//展开工位
expand_initialization_OK:=FALSE;
Expand_Group_clean_OK:=FALSE;
Expand_up_liquid_OK:=FALSE;
Expand_silica_gel_plate_OK:=FALSE;
展缸1气缸1手动:=FALSE;
展缸1气缸1自动:=FALSE;
展缸1进液电池阀1手动:=FALSE;
展缸1进液电池阀1自动:=FALSE;
展缸1排液电池阀1手动:=FALSE;
展缸1排液电池阀1自动:=FALSE;
展缸1吹气电池阀1手动:=FALSE;
展缸1吹气电池阀1自动:=FALSE;
展缸1气缸2手动:=FALSE;
展缸1气缸2自动:=FALSE;
展缸1进液电池阀2手动:=FALSE;
展缸1进液电池阀2自动:=FALSE;
展缸1排液电池阀2手动:=FALSE;
展缸1排液电池阀2自动:=FALSE;
展缸1吹气电池阀2手动:=FALSE;
展缸1吹气电池阀2自动:=FALSE;
展缸1气缸3手动:=FALSE;
展缸1气缸3自动:=FALSE;
展缸1进液电池阀3手动:=FALSE;
展缸1进液电池阀3自动:=FALSE;	
展缸1排液电池阀3手动:=FALSE;
展缸1排液电池阀3自动:=FALSE;
展缸1吹气电池阀3手动:=FALSE;
展缸1吹气电池阀3自动:=FALSE;
展缸1气缸4手动:=FALSE;
展缸1气缸4自动:=FALSE;
展缸1进液电池阀4手动:=FALSE;
展缸1进液电池阀4自动:=FALSE;	
展缸1排液电池阀4手动:=FALSE;
展缸1排液电池阀4自动:=FALSE;
展缸1吹气电池阀4手动:=FALSE;
展缸1吹气电池阀4自动:=FALSE;
展缸2气缸1手动:=FALSE;
展缸2气缸1自动:=FALSE;
展缸2进液电池阀1手动:=FALSE;
展缸2进液电池阀1自动:=FALSE;
展缸2排液电池阀1手动:=FALSE;
展缸2排液电池阀1自动:=FALSE;
展缸2吹气电池阀1手动:=FALSE;
展缸2吹气电池阀1自动:=FALSE;
展缸2气缸2手动:=FALSE;
展缸2气缸2自动:=FALSE;
展缸2进液电池阀2手动:=FALSE;
展缸2进液电池阀2自动:=FALSE;
展缸2排液电池阀2手动:=FALSE;
展缸2排液电池阀2自动:=FALSE;
展缸2吹气电池阀2手动:=FALSE;
展缸2吹气电池阀2自动:=FALSE;
展缸2气缸3手动:=FALSE;
展缸2气缸3自动:=FALSE;
展缸2进液电池阀3手动:=FALSE;
展缸2进液电池阀3自动:=FALSE;	
展缸2排液电池阀3手动:=FALSE;
展缸2排液电池阀3自动:=FALSE;
展缸2吹气电池阀3手动:=FALSE;
展缸2吹气电池阀3自动:=FALSE;
展缸2气缸4手动:=FALSE;
展缸2气缸4自动:=FALSE;
展缸2进液电池阀4手动:=FALSE;
展缸2进液电池阀4自动:=FALSE;	
展缸2排液电池阀4手动:=FALSE;
展缸2排液电池阀4自动:=FALSE;
展缸2吹气电池阀4手动:=FALSE;
展缸2吹气电池阀4自动:=FALSE;
Expand_Step:=0;
//拍照刮板
刮板拍照真空自动:=FALSE;
刮板拍照真空手动:=FALSE;
刮板拍照无刷电机手动:=FALSE;
刮板拍照无刷电机自动:=FALSE;
刮板拍照定位气缸手动:=FALSE;
刮板拍照定位气缸自动:=FALSE;
粉末收集器定位手动:=FALSE;
粉末收集器定位自动:=FALSE;
刮板拍照遮光气缸手动:=FALSE;
刮板拍照遮光气缸自动:=FALSE;
刮板拍照旋转气缸手动:=FALSE;
刮板拍照旋转气缸自动:=FALSE;
刮板拍照下压气缸手动:=FALSE;
刮板拍照下压气缸自动:=FALSE;
 scrape_IsLast := FALSE;       // ★ 新增		
scrape_PhotoMode:=0;
scrape_Step:=0;
Camera_scraper_initialization_OK:=FALSE;
Photo_preparation_completed_OK:=FALSE;
Scraper_collection_completed:=FALSE;
Robot_completes_material_retrieval:=FALSE;	

//上样点样
上样定位手动:=FALSE;
上样定位自动:=FALSE;
上样点样三通电池阀手动:=FALSE;
上样点样三通电池阀自动:=FALSE;
上样吹气手动:=FALSE;
上样吹气自动:=FALSE;
打样瓶上料轴3YDATE.fAbsTarget:=0;
点样轴6XDATE.fAbsTarget:=0;
点样轴7YDATE.fAbsTarget:=0;
上样轴4X轴DATE.fAbsTarget:=0;
上样轴5Z轴DATE.fAbsTarget:=0;
点样轴7YDATE.xMoveAbs:=FALSE;
点样轴6XDATE.xMoveAbs:=FALSE;
上样轴5Z轴DATE.xMoveAbs:=FALSE;
上样轴4X轴DATE.xMoveAbs:=FALSE;
打样瓶上料轴3YDATE.xMoveAbs:=FALSE;
Sampling_Spray_sample_OK:=FALSE;
Sampling_liquid_absorption:=FALSE;
Sampling_preparation_OK:=FALSE;
大真空泵站位[11]:=FALSE;
大真空泵自动:=FALSE;
Sampling_Step:=0;

//机器人

泵站位符:=FALSE;
上样料架报警:=FALSE;
溶液收集瓶定位自动:=FALSE;
溶液收集瓶定位手动:=FALSE;
END_ACTION

END_PROGRAM

// Device/Application/40_Man/PLC_Cyinder_气缸动作
PROGRAM PLC_Cyinder_气缸动作
VAR
	cylinder_0: FB_cylinder;
	cylinder_1: FB_cylinder;
	cylinder_2: FB_cylinder;
	cylinder_3 :FB_cylinder ;
	cylinder_4 :FB_cylinder ;
	cylinder_5 :FB_cylinder ;
	cylinder_6 :FB_cylinder ;
	cylinder_7 :FB_cylinder ;
	cylinder_8 :FB_cylinder ;
	cylinder_9 :FB_cylinder ;
	cylinder_10 :FB_cylinder ;
	cylinder_11 :FB_cylinder ;
	cylinder_12 :FB_cylinder ;
	cylinder_13 :FB_cylinder ;
	cylinder_14 :FB_cylinder ;
	cylinder_15 :FB_cylinder ;
	cylinder_16 :FB_cylinder ;
	cylinder_17 :FB_cylinder ;
	cylinder_18 :FB_cylinder ;
	cylinder_19 :FB_cylinder ;
	cylinder_20 :FB_cylinder ;
	cylinder_21 :FB_cylinder ;
	cylinder_22 :FB_cylinder ;
	cylinder_23 :FB_cylinder ;
	cylinder_24 :FB_cylinder ;
	cylinder_25 :FB_cylinder ;
	cylinder_26 :FB_cylinder ;
	cylinder_27 :FB_cylinder ;
	cylinder_28 :FB_cylinder ;
	cylinder_29 :FB_cylinder ;
	cylinder_30 :FB_cylinder ;
	cylinder_31 :FB_cylinder ;
	cylinder_32 :FB_cylinder ;
	cylinder_33 :FB_cylinder ;
	cylinder_34 :FB_cylinder ;
	cylinder_35 :FB_cylinder ;
	cylinder_36 :FB_cylinder ;
	cylinder_37 :FB_cylinder ;
	cylinder_38 :FB_cylinder ;
	cylinder_39 :FB_cylinder ;
	cylinder_40 :FB_cylinder ;
	cylinder_41 :FB_cylinder ;
	cylinder_42 :FB_cylinder ;
	cylinder_43 :FB_cylinder ;
	cylinder_44 :FB_cylinder ;
	cylinder_45 :FB_cylinder ;
	cylinder_46 :FB_cylinder ;
	cylinder_47 :FB_cylinder ;
	cylinder_48 :FB_cylinder ;
	cylinder_49 :FB_cylinder ;
	cylinder_50 :FB_cylinder ;
	bDeployCommandsArmed: BOOL;
	bAnyDeployCommandRequested: BOOL;

END_VAR

// PLC deploy auxiliary-actuator gate BEGIN
bAnyDeployCommandRequested := 展缸1气缸1手动
	OR 展缸1气缸1自动
	OR 展缸1气缸2手动
	OR 展缸1气缸2自动
	OR 展缸1气缸3手动
	OR 展缸1气缸3自动
	OR 展缸1气缸4手动
	OR 展缸1气缸4自动
	OR 展缸2气缸1手动
	OR 展缸2气缸1自动
	OR 展缸2气缸2手动
	OR 展缸2气缸2自动
	OR 展缸2气缸3手动
	OR 展缸2气缸3自动
	OR 展缸2气缸4手动
	OR 展缸2气缸4自动
	OR 大真空泵手动
	OR 大真空泵自动
	OR 收集下压气缸手动
	OR 收集下压气缸自动
	OR 收集夹持气缸手动
	OR 收集夹持气缸自动
	OR 收集升降气缸手动
	OR 收集升降气缸自动
	OR 收集伸缩气缸手动
	OR 收集伸缩气缸自动
	OR 刮板拍照遮光气缸手动
	OR 刮板拍照遮光气缸自动
	OR 刮板拍照旋转气缸手动
	OR 刮板拍照旋转气缸自动
	OR 刮板拍照下压气缸手动
	OR 刮板拍照下压气缸自动
	OR 展缸1进液电池阀1手动
	OR 展缸1进液电池阀1自动
	OR 展缸1进液电池阀2手动
	OR 展缸1进液电池阀2自动
	OR 展缸1进液电池阀3手动
	OR 展缸1进液电池阀3自动
	OR 展缸1进液电池阀4手动
	OR 展缸1进液电池阀4自动
	OR 展缸1排液电池阀1手动
	OR 展缸1排液电池阀1自动
	OR 展缸1排液电池阀2手动
	OR 展缸1排液电池阀2自动
	OR 展缸1排液电池阀3手动
	OR 展缸1排液电池阀3自动
	OR 展缸1排液电池阀4手动
	OR 展缸1排液电池阀4自动
	OR 展缸1吹气电池阀1手动
	OR 展缸1吹气电池阀1自动
	OR 展缸1吹气电池阀2手动
	OR 展缸1吹气电池阀2自动
	OR 展缸1吹气电池阀3手动
	OR 展缸1吹气电池阀3自动
	OR 展缸1吹气电池阀4手动
	OR 展缸1吹气电池阀4自动
	OR 展缸2进液电池阀1手动
	OR 展缸2进液电池阀1自动
	OR 展缸2进液电池阀2手动
	OR 展缸2进液电池阀2自动
	OR 展缸2进液电池阀3手动
	OR 展缸2进液电池阀3自动
	OR 展缸2进液电池阀4手动
	OR 展缸2进液电池阀4自动
	OR 展缸2排液电池阀1手动
	OR 展缸2排液电池阀1自动
	OR 展缸2排液电池阀2手动
	OR 展缸2排液电池阀2自动
	OR 展缸2排液电池阀3手动
	OR 展缸2排液电池阀3自动
	OR 展缸2排液电池阀4手动
	OR 展缸2排液电池阀4自动
	OR 展缸2吹气电池阀1手动
	OR 展缸2吹气电池阀1自动
	OR 展缸2吹气电池阀2手动
	OR 展缸2吹气电池阀2自动
	OR 展缸2吹气电池阀3手动
	OR 展缸2吹气电池阀3自动
	OR 展缸2吹气电池阀4手动
	OR 展缸2吹气电池阀4自动
	OR 收集进液手动
	OR 收集进液自动
	OR 收集排液手动
	OR 收集排液自动
	OR 收集正压排液手动
	OR 收集正压排液自动
	OR 溶液收集瓶定位手动
	OR 溶液收集瓶定位自动
	OR 上样定位手动
	OR 上样定位自动
	OR 上样点样三通电池阀手动
	OR 上样点样三通电池阀自动
	OR 刮板拍照真空手动
	OR 刮板拍照真空自动
	OR 刮板拍照无刷电机手动
	OR 刮板拍照无刷电机自动
	OR 刮板拍照定位气缸手动
	OR 刮板拍照定位气缸自动
	OR 粉末收集器定位手动
	OR 粉末收集器定位自动
	OR 上样吹气手动
	OR 上样吹气自动;
IF ((NOT PLC_Ready) OR ((PLC_Deploy_State<>0) AND (PLC_Deploy_State<>30))) THEN
	bDeployCommandsArmed := FALSE;
ELSIF NOT bAnyDeployCommandRequested THEN
	// A command written while maintenance was active must first return FALSE;
	// it is never replayed automatically when the maintenance lock is released.
	bDeployCommandsArmed := TRUE;
END_IF
// PLC deploy auxiliary-actuator gate END
//气缸动作
//展缸1气缸1
cylinder_0(
    xManualRetract := , 
    xAutoRetract := , 
    yValve2 => , 
    cylinder_type := 0, 

	xManualAuto:=ManualAuto  , 
	xManualExtend:=PLC_Ready AND ((PLC_Deploy_State=0) OR (PLC_Deploy_State=30)) AND bDeployCommandsArmed AND (展缸1气缸1手动), 
	xAutoExtend:= PLC_Ready AND ((PLC_Deploy_State=0) OR (PLC_Deploy_State=30)) AND bDeployCommandsArmed AND (展缸1气缸1自动), 
	xReset:=复位  , 
	xPosExtend:= 展缸1气缸1原点, 
	xPosRetract:= 展缸1气缸1动点 , 
	tTimeout:= T#5S, 
	yValve1=> 展缸1气缸1 , 
	bAlarm=> cyinderAlarm.0);
//展缸1气缸2
cylinder_1(
    xManualRetract := , 
    xAutoRetract := , 
    yValve2 => , 
    cylinder_type :=0 , 

	xManualAuto:=ManualAuto  , 
	xManualExtend:=PLC_Ready AND ((PLC_Deploy_State=0) OR (PLC_Deploy_State=30)) AND bDeployCommandsArmed AND (展缸1气缸2手动), 
	xAutoExtend:= PLC_Ready AND ((PLC_Deploy_State=0) OR (PLC_Deploy_State=30)) AND bDeployCommandsArmed AND (展缸1气缸2自动), 
	xReset:=复位  , 
	xPosExtend:= 展缸1气缸2原点, 
	xPosRetract:= 展缸1气缸2动点 , 
	tTimeout:= T#5S, 
	yValve1=> 展缸1气缸2, 
	bAlarm=> cyinderAlarm.1);
//展缸1气缸3
cylinder_2(
    xManualRetract := , 
    xAutoRetract := , 
    yValve2 => , 
    cylinder_type := 0, 

	xManualAuto:=ManualAuto  , 
	xManualExtend:=PLC_Ready AND ((PLC_Deploy_State=0) OR (PLC_Deploy_State=30)) AND bDeployCommandsArmed AND (展缸1气缸3手动), 
	xAutoExtend:= PLC_Ready AND ((PLC_Deploy_State=0) OR (PLC_Deploy_State=30)) AND bDeployCommandsArmed AND (展缸1气缸3自动), 
	xReset:=复位  , 
	xPosExtend:= 展缸1气缸3原点, 
	xPosRetract:= 展缸1气缸3动点 , 
	tTimeout:= T#5S, 
	yValve1=> 展缸1气缸3, 
	bAlarm=> cyinderAlarm.2);
//展缸1气缸4
cylinder_3(
    xManualRetract := , 
    xAutoRetract := , 
    yValve2 => , 
    cylinder_type :=0 , 

	xManualAuto:=ManualAuto  , 
	xManualExtend:=PLC_Ready AND ((PLC_Deploy_State=0) OR (PLC_Deploy_State=30)) AND bDeployCommandsArmed AND (展缸1气缸4手动), 
	xAutoExtend:= PLC_Ready AND ((PLC_Deploy_State=0) OR (PLC_Deploy_State=30)) AND bDeployCommandsArmed AND (展缸1气缸4自动), 
	xReset:=复位  , 
	xPosExtend:= 展缸1气缸4原点, 
	xPosRetract:= 展缸1气缸4动点 , 
	tTimeout:= T#5S, 
	yValve1=> 展缸1气缸4, 
	bAlarm=> cyinderAlarm.3);
//展缸2气缸1
cylinder_4(
    xManualRetract := , 
    xAutoRetract := , 
    yValve2 => , 
    cylinder_type := 0, 

	xManualAuto:=ManualAuto  , 
	xManualExtend:=PLC_Ready AND ((PLC_Deploy_State=0) OR (PLC_Deploy_State=30)) AND bDeployCommandsArmed AND (展缸2气缸1手动), 
	xAutoExtend:= PLC_Ready AND ((PLC_Deploy_State=0) OR (PLC_Deploy_State=30)) AND bDeployCommandsArmed AND (展缸2气缸1自动), 
	xReset:=复位  , 
	xPosExtend:= 展缸2气缸1原点, 
	xPosRetract:= 展缸2气缸1动点 , 
	tTimeout:= T#5S, 
	yValve1=> 展缸2气缸1, 
	bAlarm=> cyinderAlarm.4);
//展缸2气缸2
cylinder_5(
    xManualRetract := , 
    xAutoRetract := , 
    yValve2 => , 
    cylinder_type :=0 , 

	xManualAuto:=ManualAuto  , 
	xManualExtend:=PLC_Ready AND ((PLC_Deploy_State=0) OR (PLC_Deploy_State=30)) AND bDeployCommandsArmed AND (展缸2气缸2手动), 
	xAutoExtend:= PLC_Ready AND ((PLC_Deploy_State=0) OR (PLC_Deploy_State=30)) AND bDeployCommandsArmed AND (展缸2气缸2自动), 
	xReset:=复位  , 
	xPosExtend:= 展缸2气缸2原点, 
	xPosRetract:= 展缸2气缸2动点 , 
	tTimeout:= T#5S, 
	yValve1=> 展缸2气缸2, 
	bAlarm=> cyinderAlarm.5);
//展缸2气缸3
cylinder_6(
    xManualRetract := , 
    xAutoRetract := , 
    yValve2 => , 
    cylinder_type := 0, 

	xManualAuto:=ManualAuto  , 
	xManualExtend:=PLC_Ready AND ((PLC_Deploy_State=0) OR (PLC_Deploy_State=30)) AND bDeployCommandsArmed AND (展缸2气缸3手动), 
	xAutoExtend:= PLC_Ready AND ((PLC_Deploy_State=0) OR (PLC_Deploy_State=30)) AND bDeployCommandsArmed AND (展缸2气缸3自动), 
	xReset:=复位  , 
	xPosExtend:= 展缸2气缸3原点, 
	xPosRetract:= 展缸2气缸3动点 , 
	tTimeout:= T#5S, 
	yValve1=> 展缸2气缸3, 
	bAlarm=> cyinderAlarm.6);
//展缸2气缸4
cylinder_7(
    xManualRetract := , 
    xAutoRetract := , 
    yValve2 => , 
    cylinder_type := 0, 

	xManualAuto:=ManualAuto  , 
	xManualExtend:=PLC_Ready AND ((PLC_Deploy_State=0) OR (PLC_Deploy_State=30)) AND bDeployCommandsArmed AND (展缸2气缸4手动), 
	xAutoExtend:= PLC_Ready AND ((PLC_Deploy_State=0) OR (PLC_Deploy_State=30)) AND bDeployCommandsArmed AND (展缸2气缸4自动), 
	xReset:=复位  , 
	xPosExtend:= 展缸2气缸4原点, 
	xPosRetract:= 展缸2气缸4动点 , 
	tTimeout:= T#5S, 
	yValve1=> 展缸2气缸4, 
	bAlarm=> cyinderAlarm.7);
//大真空泵
cylinder_8(
    xManualRetract := , 
    xAutoRetract := , 
    yValve2 => , 
    cylinder_type :=0 , 

	xManualAuto:=ManualAuto  , 
	xManualExtend:= PLC_Ready AND ((PLC_Deploy_State=0) OR (PLC_Deploy_State=30)) AND bDeployCommandsArmed AND (大真空泵手动), 
	xAutoExtend:= PLC_Ready AND ((PLC_Deploy_State=0) OR (PLC_Deploy_State=30)) AND bDeployCommandsArmed AND (大真空泵自动), 
	xReset:=复位  , 
	xPosExtend:= , 
	xPosRetract:=  , 
	tTimeout:= , 
	yValve1=> 大真空泵, 
	bAlarm=> );
//收集平台下压气缸
cylinder_9(
    xManualRetract := , 
    xAutoRetract := , 
    yValve2 => , 
    cylinder_type := 0, 

	xManualAuto:=ManualAuto  , 
	xManualExtend:= PLC_Ready AND ((PLC_Deploy_State=0) OR (PLC_Deploy_State=30)) AND bDeployCommandsArmed AND (收集下压气缸手动), 
	xAutoExtend:= PLC_Ready AND ((PLC_Deploy_State=0) OR (PLC_Deploy_State=30)) AND bDeployCommandsArmed AND (收集下压气缸自动), 
	xReset:=复位  , 
	xPosExtend:=收集平台下压气缸原点 , 
	xPosRetract:= 收集下压气缸手动 OR 收集下压气缸自动, 
	tTimeout:= T#5S, 
	yValve1=> 收集下压气缸 , 
	bAlarm=> cyinderAlarm.8);
//收集平台夹持气缸
cylinder_10(
    xManualRetract := , 
    xAutoRetract := , 
    yValve2 => , 
    cylinder_type := 0, 

	xManualAuto:=ManualAuto  , 
	xManualExtend:= PLC_Ready AND ((PLC_Deploy_State=0) OR (PLC_Deploy_State=30)) AND bDeployCommandsArmed AND (收集夹持气缸手动), 
	xAutoExtend:= PLC_Ready AND ((PLC_Deploy_State=0) OR (PLC_Deploy_State=30)) AND bDeployCommandsArmed AND (收集夹持气缸自动), 
	xReset:=复位  , 
	xPosExtend:=收集平台夹持气缸原点 , 
	xPosRetract:= 收集平台夹持气缸动点, 
	tTimeout:= T#5S, 
	yValve1=> 收集夹持气缸  , 
	bAlarm=> cyinderAlarm.9);	
//收集平台升降气缸
cylinder_11(
    xManualRetract := , 
    xAutoRetract := , 
    yValve2 => , 
    cylinder_type := 0, 

	xManualAuto:=ManualAuto  , 
	xManualExtend:= PLC_Ready AND ((PLC_Deploy_State=0) OR (PLC_Deploy_State=30)) AND bDeployCommandsArmed AND (收集升降气缸手动), 
	xAutoExtend:= PLC_Ready AND ((PLC_Deploy_State=0) OR (PLC_Deploy_State=30)) AND bDeployCommandsArmed AND (收集升降气缸自动), 
	xReset:=复位  , 
	xPosExtend:=收集平台升降气缸原点 , 
	xPosRetract:= 收集平台升降气缸动点, 
	tTimeout:= T#5S, 
	yValve1=> 收集升降气缸   , 
	bAlarm=> cyinderAlarm.10);	
//收集平台伸缩气缸
cylinder_12(
    xManualRetract := , 
    xAutoRetract := , 
    yValve2 => , 
    cylinder_type :=0 , 

	xManualAuto:=ManualAuto  , 
	xManualExtend:= PLC_Ready AND ((PLC_Deploy_State=0) OR (PLC_Deploy_State=30)) AND bDeployCommandsArmed AND (收集伸缩气缸手动), 
	xAutoExtend:= PLC_Ready AND ((PLC_Deploy_State=0) OR (PLC_Deploy_State=30)) AND bDeployCommandsArmed AND (收集伸缩气缸自动), 
	xReset:=复位, 
	xPosExtend:=收集平台推出气缸原点, 
	xPosRetract:= 收集平台推出气缸动点, 
	tTimeout:= T#5S, 
	yValve1=> 收集伸缩气缸, 
	bAlarm=> cyinderAlarm.11);		
//刮板拍照遮光气缸
cylinder_13(
    xManualRetract := , 
    xAutoRetract := , 
    yValve2 => , 
    cylinder_type :=0 , 

	xManualAuto:=ManualAuto  , 
	xManualExtend:= PLC_Ready AND ((PLC_Deploy_State=0) OR (PLC_Deploy_State=30)) AND bDeployCommandsArmed AND (刮板拍照遮光气缸手动), 
	xAutoExtend:=PLC_Ready AND ((PLC_Deploy_State=0) OR (PLC_Deploy_State=30)) AND bDeployCommandsArmed AND (刮板拍照遮光气缸自动), 
	xReset:=复位  , 
	xPosExtend:=刮板拍照遮光气缸上位 , 
	xPosRetract:= 刮板拍照遮光气缸下位, 
	tTimeout:= T#5S, 
	yValve1=>  刮板拍照遮光气缸, 
	bAlarm=> cyinderAlarm.12);		
//刮板拍照旋转气缸
cylinder_14(
    xManualRetract := , 
    xAutoRetract := , 
    yValve2 => , 
    cylinder_type := 0, 

	xManualAuto:=ManualAuto  , 
	xManualExtend:= PLC_Ready AND ((PLC_Deploy_State=0) OR (PLC_Deploy_State=30)) AND bDeployCommandsArmed AND (刮板拍照旋转气缸手动 AND 刮板轴9XDATE.fActPos>330), 
	xAutoExtend:=PLC_Ready AND ((PLC_Deploy_State=0) OR (PLC_Deploy_State=30)) AND bDeployCommandsArmed AND (刮板拍照旋转气缸自动), 
	xReset:=复位  , 
	xPosExtend:=刮板拍照旋转气缸原点  , 
	xPosRetract:= 刮板拍照旋转气缸动点, 
	tTimeout:= T#5S, 
	yValve1=>  刮板拍照旋转气缸   , 
	bAlarm=> cyinderAlarm.13);		
//刮板拍照下压气缸
cylinder_15(
    xManualRetract := , 
    xAutoRetract := , 
    yValve2 => , 
    cylinder_type := 0, 

	xManualAuto:=ManualAuto  , 
	xManualExtend:= PLC_Ready AND ((PLC_Deploy_State=0) OR (PLC_Deploy_State=30)) AND bDeployCommandsArmed AND (刮板拍照下压气缸手动), 
	xAutoExtend:=PLC_Ready AND ((PLC_Deploy_State=0) OR (PLC_Deploy_State=30)) AND bDeployCommandsArmed AND (刮板拍照下压气缸自动), 
	xReset:=复位  , 
	xPosExtend:=刮板拍照下压气缸上位, 
	xPosRetract:=刮板拍照下压气缸手动 OR 刮板拍照下压气缸自动 , 
	tTimeout:= T#5S, 
	yValve1=>  刮板拍照下压气缸, 
	bAlarm=> cyinderAlarm.14);
//展缸1进液电池阀1
cylinder_17(
    xManualRetract := , 
    xAutoRetract := , 
    yValve2 => , 
    cylinder_type :=0 , 

	xManualAuto:=ManualAuto  , 
	xManualExtend:= PLC_Ready AND ((PLC_Deploy_State=0) OR (PLC_Deploy_State=30)) AND bDeployCommandsArmed AND (展缸1进液电池阀1手动), 
	xAutoExtend:= PLC_Ready AND ((PLC_Deploy_State=0) OR (PLC_Deploy_State=30)) AND bDeployCommandsArmed AND (展缸1进液电池阀1自动), 
	xReset:=复位  , 
	xPosExtend:=   , 
	xPosRetract:= , 
	tTimeout:= , 
	yValve1=> 展缸1进液电池阀1, 
	bAlarm=> );	
//展缸1进液电池阀2
cylinder_18(
    xManualRetract := , 
    xAutoRetract := , 
    yValve2 => , 
    cylinder_type := 0, 

	xManualAuto:=ManualAuto  , 
	xManualExtend:= PLC_Ready AND ((PLC_Deploy_State=0) OR (PLC_Deploy_State=30)) AND bDeployCommandsArmed AND (展缸1进液电池阀2手动), 
	xAutoExtend:= PLC_Ready AND ((PLC_Deploy_State=0) OR (PLC_Deploy_State=30)) AND bDeployCommandsArmed AND (展缸1进液电池阀2自动), 
	xReset:=复位  , 
	xPosExtend:=   , 
	xPosRetract:= , 
	tTimeout:= , 
	yValve1=> 展缸1进液电池阀2, 
	bAlarm=> );	
//展缸1进液电池阀3
cylinder_19(
    xManualRetract := , 
    xAutoRetract := , 
    yValve2 => , 
    cylinder_type := 0, 

	xManualAuto:=ManualAuto  , 
	xManualExtend:= PLC_Ready AND ((PLC_Deploy_State=0) OR (PLC_Deploy_State=30)) AND bDeployCommandsArmed AND (展缸1进液电池阀3手动), 
	xAutoExtend:= PLC_Ready AND ((PLC_Deploy_State=0) OR (PLC_Deploy_State=30)) AND bDeployCommandsArmed AND (展缸1进液电池阀3自动), 
	xReset:=复位  , 
	xPosExtend:=   , 
	xPosRetract:= , 
	tTimeout:= , 
	yValve1=> 展缸1进液电池阀3, 
	bAlarm=> );	
//展缸1进液电池阀4
cylinder_20(
    xManualRetract := , 
    xAutoRetract := , 
    yValve2 => , 
    cylinder_type := 0, 

	xManualAuto:=ManualAuto  , 
	xManualExtend:= PLC_Ready AND ((PLC_Deploy_State=0) OR (PLC_Deploy_State=30)) AND bDeployCommandsArmed AND (展缸1进液电池阀4手动), 
	xAutoExtend:= PLC_Ready AND ((PLC_Deploy_State=0) OR (PLC_Deploy_State=30)) AND bDeployCommandsArmed AND (展缸1进液电池阀4自动), 
	xReset:=复位  , 
	xPosExtend:=   , 
	xPosRetract:= , 
	tTimeout:= , 
	yValve1=> 展缸1进液电池阀4, 
	bAlarm=> );	
//展缸1排液电池阀1
cylinder_21(
    xManualRetract := , 
    xAutoRetract := , 
    yValve2 => , 
    cylinder_type := 0, 

	xManualAuto:=ManualAuto  , 
	xManualExtend:= PLC_Ready AND ((PLC_Deploy_State=0) OR (PLC_Deploy_State=30)) AND bDeployCommandsArmed AND (展缸1排液电池阀1手动), 
	xAutoExtend:= PLC_Ready AND ((PLC_Deploy_State=0) OR (PLC_Deploy_State=30)) AND bDeployCommandsArmed AND (展缸1排液电池阀1自动), 
	xReset:=复位  , 
	xPosExtend:=   , 
	xPosRetract:= , 
	tTimeout:= , 
	yValve1=> 展缸1排液电池阀1, 
	bAlarm=> );	
//展缸1排液电池阀2
cylinder_22(
    xManualRetract := , 
    xAutoRetract := , 
    yValve2 => , 
    cylinder_type :=0 , 

	xManualAuto:=ManualAuto  , 
	xManualExtend:= PLC_Ready AND ((PLC_Deploy_State=0) OR (PLC_Deploy_State=30)) AND bDeployCommandsArmed AND (展缸1排液电池阀2手动), 
	xAutoExtend:= PLC_Ready AND ((PLC_Deploy_State=0) OR (PLC_Deploy_State=30)) AND bDeployCommandsArmed AND (展缸1排液电池阀2自动), 
	xReset:=复位  , 
	xPosExtend:=   , 
	xPosRetract:= , 
	tTimeout:= , 
	yValve1=> 展缸1排液电池阀2, 
	bAlarm=> );	
//展缸1排液电池阀3
cylinder_23(
    xManualRetract := , 
    xAutoRetract := , 
    yValve2 => , 
    cylinder_type :=0 , 

	xManualAuto:=ManualAuto, 
	xManualExtend:= PLC_Ready AND ((PLC_Deploy_State=0) OR (PLC_Deploy_State=30)) AND bDeployCommandsArmed AND (展缸1排液电池阀3手动), 
	xAutoExtend:= PLC_Ready AND ((PLC_Deploy_State=0) OR (PLC_Deploy_State=30)) AND bDeployCommandsArmed AND (展缸1排液电池阀3自动), 
	xReset:=复位  , 
	xPosExtend:=   , 
	xPosRetract:= , 
	tTimeout:= , 
	yValve1=> 展缸1排液电池阀3, 
	bAlarm=> );	
//展缸1排液电池阀4
cylinder_24(
    xManualRetract := , 
    xAutoRetract := , 
    yValve2 => , 
    cylinder_type := 0, 

	xManualAuto:=ManualAuto, 
	xManualExtend:= PLC_Ready AND ((PLC_Deploy_State=0) OR (PLC_Deploy_State=30)) AND bDeployCommandsArmed AND (展缸1排液电池阀4手动), 
	xAutoExtend:= PLC_Ready AND ((PLC_Deploy_State=0) OR (PLC_Deploy_State=30)) AND bDeployCommandsArmed AND (展缸1排液电池阀4自动), 
	xReset:=复位  , 
	xPosExtend:=   , 
	xPosRetract:= , 
	tTimeout:= , 
	yValve1=> 展缸1排液电池阀4, 
	bAlarm=> );	
//展缸1吹气电池阀1
cylinder_25(
    xManualRetract := , 
    xAutoRetract := , 
    yValve2 => , 
    cylinder_type := 0, 

	xManualAuto:=ManualAuto, 
	xManualExtend:= PLC_Ready AND ((PLC_Deploy_State=0) OR (PLC_Deploy_State=30)) AND bDeployCommandsArmed AND (展缸1吹气电池阀1手动), 
	xAutoExtend:= PLC_Ready AND ((PLC_Deploy_State=0) OR (PLC_Deploy_State=30)) AND bDeployCommandsArmed AND (展缸1吹气电池阀1自动), 
	xReset:=复位  , 
	xPosExtend:=   , 
	xPosRetract:= , 
	tTimeout:= , 
	yValve1=> 展缸1吹气电池阀1, 
	bAlarm=> );	
//展缸1吹气电池阀2
cylinder_26(
    xManualRetract := , 
    xAutoRetract := , 
    yValve2 => , 
    cylinder_type := 0, 

	xManualAuto:=ManualAuto, 
	xManualExtend:= PLC_Ready AND ((PLC_Deploy_State=0) OR (PLC_Deploy_State=30)) AND bDeployCommandsArmed AND (展缸1吹气电池阀2手动), 
	xAutoExtend:= PLC_Ready AND ((PLC_Deploy_State=0) OR (PLC_Deploy_State=30)) AND bDeployCommandsArmed AND (展缸1吹气电池阀2自动), 
	xReset:=复位  , 
	xPosExtend:=   , 
	xPosRetract:= , 
	tTimeout:= , 
	yValve1=> 展缸1吹气电池阀2, 
	bAlarm=> );	
//展缸1吹气电池阀3
cylinder_27(
    xManualRetract := , 
    xAutoRetract := , 
    yValve2 => , 
    cylinder_type := 0, 

	xManualAuto:=ManualAuto  , 
	xManualExtend:= PLC_Ready AND ((PLC_Deploy_State=0) OR (PLC_Deploy_State=30)) AND bDeployCommandsArmed AND (展缸1吹气电池阀3手动), 
	xAutoExtend:= PLC_Ready AND ((PLC_Deploy_State=0) OR (PLC_Deploy_State=30)) AND bDeployCommandsArmed AND (展缸1吹气电池阀3自动), 
	xReset:=复位  , 
	xPosExtend:=   , 
	xPosRetract:= , 
	tTimeout:= , 
	yValve1=> 展缸1吹气电池阀3, 
	bAlarm=> );	
//展缸1吹气电池阀4
cylinder_28(
    xManualRetract := , 
    xAutoRetract := , 
    yValve2 => , 
    cylinder_type := 0, 

	xManualAuto:=ManualAuto, 
	xManualExtend:= PLC_Ready AND ((PLC_Deploy_State=0) OR (PLC_Deploy_State=30)) AND bDeployCommandsArmed AND (展缸1吹气电池阀4手动), 
	xAutoExtend:= PLC_Ready AND ((PLC_Deploy_State=0) OR (PLC_Deploy_State=30)) AND bDeployCommandsArmed AND (展缸1吹气电池阀4自动), 
	xReset:=复位  , 
	xPosExtend:=   , 
	xPosRetract:= , 
	tTimeout:= , 
	yValve1=> 展缸1吹气电池阀4, 
	bAlarm=> );	
//展缸2进液电池阀1
cylinder_29(
    xManualRetract := , 
    xAutoRetract := , 
    yValve2 => , 
    cylinder_type := 0, 

	xManualAuto:=ManualAuto, 
	xManualExtend:= PLC_Ready AND ((PLC_Deploy_State=0) OR (PLC_Deploy_State=30)) AND bDeployCommandsArmed AND (展缸2进液电池阀1手动), 
	xAutoExtend:= PLC_Ready AND ((PLC_Deploy_State=0) OR (PLC_Deploy_State=30)) AND bDeployCommandsArmed AND (展缸2进液电池阀1自动), 
	xReset:=复位  , 
	xPosExtend:=   , 
	xPosRetract:= , 
	tTimeout:= , 
	yValve1=> 展缸2进液电池阀1, 
	bAlarm=> );	
//展缸2进液电池阀2
cylinder_30(
    xManualRetract := , 
    xAutoRetract := , 
    yValve2 => , 
    cylinder_type := 0, 

	xManualAuto:=ManualAuto, 
	xManualExtend:= PLC_Ready AND ((PLC_Deploy_State=0) OR (PLC_Deploy_State=30)) AND bDeployCommandsArmed AND (展缸2进液电池阀2手动), 
	xAutoExtend:= PLC_Ready AND ((PLC_Deploy_State=0) OR (PLC_Deploy_State=30)) AND bDeployCommandsArmed AND (展缸2进液电池阀2自动), 
	xReset:=复位  , 
	xPosExtend:=   , 
	xPosRetract:= , 
	tTimeout:= , 
	yValve1=> 展缸2进液电池阀2, 
	bAlarm=> );	
//展缸2进液电池阀3
cylinder_31(
    xManualRetract := , 
    xAutoRetract := , 
    yValve2 => , 
    cylinder_type := 0, 

	xManualAuto:=ManualAuto, 
	xManualExtend:= PLC_Ready AND ((PLC_Deploy_State=0) OR (PLC_Deploy_State=30)) AND bDeployCommandsArmed AND (展缸2进液电池阀3手动), 
	xAutoExtend:= PLC_Ready AND ((PLC_Deploy_State=0) OR (PLC_Deploy_State=30)) AND bDeployCommandsArmed AND (展缸2进液电池阀3自动), 
	xReset:=复位  , 
	xPosExtend:=   , 
	xPosRetract:= , 
	tTimeout:= , 
	yValve1=> 展缸2进液电池阀3, 
	bAlarm=> );	
//展缸2进液电池阀4
cylinder_32(
    xManualRetract := , 
    xAutoRetract := , 
    yValve2 => , 
    cylinder_type := 0, 

	xManualAuto:=ManualAuto, 
	xManualExtend:= PLC_Ready AND ((PLC_Deploy_State=0) OR (PLC_Deploy_State=30)) AND bDeployCommandsArmed AND (展缸2进液电池阀4手动), 
	xAutoExtend:= PLC_Ready AND ((PLC_Deploy_State=0) OR (PLC_Deploy_State=30)) AND bDeployCommandsArmed AND (展缸2进液电池阀4自动), 
	xReset:=复位  , 
	xPosExtend:=   , 
	xPosRetract:= , 
	tTimeout:= , 
	yValve1=> 展缸2进液电池阀4, 
	bAlarm=> );	
//展缸2排液电池阀1
cylinder_33(
    xManualRetract := , 
    xAutoRetract := , 
    yValve2 => , 
    cylinder_type := 0, 

	xManualAuto:=ManualAuto, 
	xManualExtend:= PLC_Ready AND ((PLC_Deploy_State=0) OR (PLC_Deploy_State=30)) AND bDeployCommandsArmed AND (展缸2排液电池阀1手动), 
	xAutoExtend:= PLC_Ready AND ((PLC_Deploy_State=0) OR (PLC_Deploy_State=30)) AND bDeployCommandsArmed AND (展缸2排液电池阀1自动), 
	xReset:=复位  , 
	xPosExtend:=   , 
	xPosRetract:= , 
	tTimeout:= , 
	yValve1=> 展缸2排液电池阀1, 
	bAlarm=> );	
//展缸2排液电池阀2
cylinder_34(
    xManualRetract := , 
    xAutoRetract := , 
    yValve2 => , 
    cylinder_type := 0, 

	xManualAuto:=ManualAuto, 
	xManualExtend:= PLC_Ready AND ((PLC_Deploy_State=0) OR (PLC_Deploy_State=30)) AND bDeployCommandsArmed AND (展缸2排液电池阀2手动), 
	xAutoExtend:= PLC_Ready AND ((PLC_Deploy_State=0) OR (PLC_Deploy_State=30)) AND bDeployCommandsArmed AND (展缸2排液电池阀2自动), 
	xReset:=复位  , 
	xPosExtend:=   , 
	xPosRetract:= , 
	tTimeout:= , 
	yValve1=> 展缸2排液电池阀2, 
	bAlarm=> );	
//展缸2排液电池阀3
cylinder_35(
    xManualRetract := , 
    xAutoRetract := , 
    yValve2 => , 
    cylinder_type := 0, 

	xManualAuto:=ManualAuto, 
	xManualExtend:= PLC_Ready AND ((PLC_Deploy_State=0) OR (PLC_Deploy_State=30)) AND bDeployCommandsArmed AND (展缸2排液电池阀3手动), 
	xAutoExtend:= PLC_Ready AND ((PLC_Deploy_State=0) OR (PLC_Deploy_State=30)) AND bDeployCommandsArmed AND (展缸2排液电池阀3自动), 
	xReset:=复位  , 
	xPosExtend:=   , 
	xPosRetract:= , 
	tTimeout:= , 
	yValve1=> 展缸2排液电池阀3, 
	bAlarm=> );	
//展缸2排液电池阀4
cylinder_36(
    xManualRetract := , 
    xAutoRetract := , 
    yValve2 => , 
    cylinder_type :=0 , 

	xManualAuto:=ManualAuto, 
	xManualExtend:= PLC_Ready AND ((PLC_Deploy_State=0) OR (PLC_Deploy_State=30)) AND bDeployCommandsArmed AND (展缸2排液电池阀4手动), 
	xAutoExtend:= PLC_Ready AND ((PLC_Deploy_State=0) OR (PLC_Deploy_State=30)) AND bDeployCommandsArmed AND (展缸2排液电池阀4自动), 
	xReset:=复位  , 
	xPosExtend:=   , 
	xPosRetract:= , 
	tTimeout:= , 
	yValve1=> 展缸2排液电池阀4, 
	bAlarm=> );	
//展缸2吹气电池阀1
cylinder_37(
    xManualRetract := , 
    xAutoRetract := , 
    yValve2 => , 
    cylinder_type := 0, 

	xManualAuto:=ManualAuto, 
	xManualExtend:= PLC_Ready AND ((PLC_Deploy_State=0) OR (PLC_Deploy_State=30)) AND bDeployCommandsArmed AND (展缸2吹气电池阀1手动), 
	xAutoExtend:= PLC_Ready AND ((PLC_Deploy_State=0) OR (PLC_Deploy_State=30)) AND bDeployCommandsArmed AND (展缸2吹气电池阀1自动), 
	xReset:=复位  , 
	xPosExtend:=   , 
	xPosRetract:= , 
	tTimeout:= , 
	yValve1=> 展缸2吹气电池阀1, 
	bAlarm=> );	
//展缸2吹气电池阀2
cylinder_38(
    xManualRetract := , 
    xAutoRetract := , 
    yValve2 => , 
    cylinder_type := 0, 

	xManualAuto:=ManualAuto, 
	xManualExtend:= PLC_Ready AND ((PLC_Deploy_State=0) OR (PLC_Deploy_State=30)) AND bDeployCommandsArmed AND (展缸2吹气电池阀2手动), 
	xAutoExtend:= PLC_Ready AND ((PLC_Deploy_State=0) OR (PLC_Deploy_State=30)) AND bDeployCommandsArmed AND (展缸2吹气电池阀2自动), 
	xReset:=复位  , 
	xPosExtend:=   , 
	xPosRetract:= , 
	tTimeout:= , 
	yValve1=> 展缸2吹气电池阀2, 
	bAlarm=> );	
//展缸1吹气电池阀3
cylinder_39(
    xManualRetract := , 
    xAutoRetract := , 
    yValve2 => , 
    cylinder_type := 0, 

	xManualAuto:=ManualAuto, 
	xManualExtend:= PLC_Ready AND ((PLC_Deploy_State=0) OR (PLC_Deploy_State=30)) AND bDeployCommandsArmed AND (展缸2吹气电池阀3手动), 
	xAutoExtend:= PLC_Ready AND ((PLC_Deploy_State=0) OR (PLC_Deploy_State=30)) AND bDeployCommandsArmed AND (展缸2吹气电池阀3自动), 
	xReset:=复位  , 
	xPosExtend:=   , 
	xPosRetract:= , 
	tTimeout:= , 
	yValve1=> 展缸2吹气电池阀3, 
	bAlarm=> );	
//展缸2吹气电池阀4
cylinder_40(
    xManualRetract := , 
    xAutoRetract := , 
    yValve2 => , 
    cylinder_type := 0, 

	xManualAuto:=ManualAuto, 
	xManualExtend:= PLC_Ready AND ((PLC_Deploy_State=0) OR (PLC_Deploy_State=30)) AND bDeployCommandsArmed AND (展缸2吹气电池阀4手动), 
	xAutoExtend:= PLC_Ready AND ((PLC_Deploy_State=0) OR (PLC_Deploy_State=30)) AND bDeployCommandsArmed AND (展缸2吹气电池阀4自动), 
	xReset:=复位  , 
	xPosExtend:=   , 
	xPosRetract:= , 
	tTimeout:= , 
	yValve1=> 展缸2吹气电池阀4, 
	bAlarm=> );	
//收集进液电池阀
cylinder_41(
    xManualRetract := , 
    xAutoRetract := , 
    yValve2 => , 
    cylinder_type := 0, 

	xManualAuto:=ManualAuto, 
	xManualExtend:= PLC_Ready AND ((PLC_Deploy_State=0) OR (PLC_Deploy_State=30)) AND bDeployCommandsArmed AND (收集进液手动), 
	xAutoExtend:= PLC_Ready AND ((PLC_Deploy_State=0) OR (PLC_Deploy_State=30)) AND bDeployCommandsArmed AND (收集进液自动), 
	xReset:=复位  , 
	xPosExtend:=   , 
	xPosRetract:= , 
	tTimeout:= , 
	yValve1=> 收集平台进液2通电池阀, 
	bAlarm=> );	
//收集排液电池阀
cylinder_42(
    xManualRetract := , 
    xAutoRetract := , 
    yValve2 => , 
    cylinder_type := 0, 

	xManualAuto:=ManualAuto  , 
	xManualExtend:= PLC_Ready AND ((PLC_Deploy_State=0) OR (PLC_Deploy_State=30)) AND bDeployCommandsArmed AND (收集排液手动), 
	xAutoExtend:= PLC_Ready AND ((PLC_Deploy_State=0) OR (PLC_Deploy_State=30)) AND bDeployCommandsArmed AND (收集排液自动), 
	xReset:=复位  , 
	xPosExtend:=   , 
	xPosRetract:= , 
	tTimeout:= , 
	yValve1=> 收集平台排液3通电池阀, 
	bAlarm=> );	
//收集正压排液电池阀
cylinder_43(
    xManualRetract := , 
    xAutoRetract := , 
    yValve2 => , 
    cylinder_type :=0 , 

	xManualAuto:=ManualAuto  , 
	xManualExtend:= PLC_Ready AND ((PLC_Deploy_State=0) OR (PLC_Deploy_State=30)) AND bDeployCommandsArmed AND (收集正压排液手动), 
	xAutoExtend:= PLC_Ready AND ((PLC_Deploy_State=0) OR (PLC_Deploy_State=30)) AND bDeployCommandsArmed AND (收集正压排液自动), 
	xReset:=复位  , 
	xPosExtend:=   , 
	xPosRetract:= , 
	tTimeout:= , 
	yValve1=> 收集平台正压排液阀, 
	bAlarm=> );	
//溶液收集瓶定位气缸
cylinder_44(
    xManualRetract := , 
    xAutoRetract := , 
    yValve2 => , 
    cylinder_type := 0, 

	xManualAuto:=ManualAuto  , 
	xManualExtend:= PLC_Ready AND ((PLC_Deploy_State=0) OR (PLC_Deploy_State=30)) AND bDeployCommandsArmed AND (溶液收集瓶定位手动), 
	xAutoExtend:= PLC_Ready AND ((PLC_Deploy_State=0) OR (PLC_Deploy_State=30)) AND bDeployCommandsArmed AND (溶液收集瓶定位自动), 
	xReset:=复位  , 
	xPosExtend:=   , 
	xPosRetract:= , 
	tTimeout:= , 
	yValve1=> 溶液收集瓶工位定位气缸, 
	bAlarm=> );	
//上样定位气缸
cylinder_45(
    xManualRetract := , 
    xAutoRetract := , 
    yValve2 => , 
    cylinder_type :=0 , 

	xManualAuto:=ManualAuto  , 
	xManualExtend:= PLC_Ready AND ((PLC_Deploy_State=0) OR (PLC_Deploy_State=30)) AND bDeployCommandsArmed AND (上样定位手动), 
	xAutoExtend:= PLC_Ready AND ((PLC_Deploy_State=0) OR (PLC_Deploy_State=30)) AND bDeployCommandsArmed AND (上样定位自动), 
	xReset:=复位  , 
	xPosExtend:=   , 
	xPosRetract:= , 
	tTimeout:= , 
	yValve1=> 上样定位气缸, 
	bAlarm=> );	
//上样点样三通电池阀
cylinder_46(
    xManualRetract := , 
    xAutoRetract := , 
    yValve2 => , 
    cylinder_type :=0 , 

	xManualAuto:=ManualAuto  , 
	xManualExtend:= PLC_Ready AND ((PLC_Deploy_State=0) OR (PLC_Deploy_State=30)) AND bDeployCommandsArmed AND (上样点样三通电池阀手动), 
	xAutoExtend:= PLC_Ready AND ((PLC_Deploy_State=0) OR (PLC_Deploy_State=30)) AND bDeployCommandsArmed AND (上样点样三通电池阀自动), 
	xReset:=复位  , 
	xPosExtend:=   , 
	xPosRetract:= , 
	tTimeout:= , 
	yValve1=> 上样点样三通电池阀, 
	bAlarm=> );	
//刮板拍照真空泵
cylinder_46(
    xManualRetract := , 
    xAutoRetract := , 
    yValve2 => , 
    cylinder_type := 0, 

	xManualAuto:=ManualAuto  , 
	xManualExtend:=PLC_Ready AND ((PLC_Deploy_State=0) OR (PLC_Deploy_State=30)) AND bDeployCommandsArmed AND (刮板拍照真空手动), 
	xAutoExtend:= PLC_Ready AND ((PLC_Deploy_State=0) OR (PLC_Deploy_State=30)) AND bDeployCommandsArmed AND (刮板拍照真空自动), 
	xReset:=复位  , 
	xPosExtend:=   , 
	xPosRetract:= , 
	tTimeout:= , 
	yValve1=> 刮板拍照真空阀, 
	bAlarm=> );	
//刮板拍照无刷电机
cylinder_47(
    xManualRetract := , 
    xAutoRetract := , 
    yValve2 => , 
    cylinder_type :=0 , 

	xManualAuto:=ManualAuto  , 
	xManualExtend:=PLC_Ready AND ((PLC_Deploy_State=0) OR (PLC_Deploy_State=30)) AND bDeployCommandsArmed AND (刮板拍照无刷电机手动), 
	xAutoExtend:=PLC_Ready AND ((PLC_Deploy_State=0) OR (PLC_Deploy_State=30)) AND bDeployCommandsArmed AND (刮板拍照无刷电机自动), 
	xReset:=复位  , 
	xPosExtend:=   , 
	xPosRetract:= , 
	tTimeout:= , 
	yValve1=> 刮板拍照无刷电机, 
	bAlarm=> );	
//刮板拍照定位气缸
cylinder_48(
    xManualRetract := , 
    xAutoRetract := , 
    yValve2 => , 
    cylinder_type :=0 , 

	xManualAuto:=ManualAuto  , 
	xManualExtend:= PLC_Ready AND ((PLC_Deploy_State=0) OR (PLC_Deploy_State=30)) AND bDeployCommandsArmed AND (刮板拍照定位气缸手动), 
	xAutoExtend:=PLC_Ready AND ((PLC_Deploy_State=0) OR (PLC_Deploy_State=30)) AND bDeployCommandsArmed AND (刮板拍照定位气缸自动), 
	xReset:=复位  , 
	xPosExtend:=   , 
	xPosRetract:= , 
	tTimeout:= , 
	yValve1=> 刮板拍照定位气缸, 
	bAlarm=> );	
//粉末收集器定位气缸
cylinder_49(
    xManualRetract := , 
    xAutoRetract := , 
    yValve2 => , 
    cylinder_type :=0 , 

	xManualAuto:=ManualAuto  , 
	xManualExtend:= PLC_Ready AND ((PLC_Deploy_State=0) OR (PLC_Deploy_State=30)) AND bDeployCommandsArmed AND (粉末收集器定位手动), 
	xAutoExtend:= PLC_Ready AND ((PLC_Deploy_State=0) OR (PLC_Deploy_State=30)) AND bDeployCommandsArmed AND (粉末收集器定位自动), 
	xReset:=复位  , 
	xPosExtend:=   , 
	xPosRetract:= , 
	tTimeout:= , 
	yValve1=> 粉末收集器工位定位气缸, 
	bAlarm=> );	
//上样吹气电池阀
cylinder_50(
    xManualRetract := , 
    xAutoRetract := , 
    yValve2 => , 
    cylinder_type := 0, 

	xManualAuto:=ManualAuto  , 
	xManualExtend:= PLC_Ready AND ((PLC_Deploy_State=0) OR (PLC_Deploy_State=30)) AND bDeployCommandsArmed AND (上样吹气手动), 
	xAutoExtend:= PLC_Ready AND ((PLC_Deploy_State=0) OR (PLC_Deploy_State=30)) AND bDeployCommandsArmed AND (上样吹气自动), 
	xReset:=复位  , 
	xPosExtend:=   , 
	xPosRetract:= , 
	tTimeout:= , 
	yValve1=> 上样吹气二通阀, 
	bAlarm=> );

END_PROGRAM

// Device/Application/25_FB_功能块/FB_cylinder
FUNCTION_BLOCK FB_cylinder
VAR_INPUT
    xManualAuto : BOOL := FALSE;  // 手自动模式：FALSE=手动，TRUE=自动
    xManualExtend : BOOL;  // 手动伸出
	// 手动缩回
	xManualRetract: BOOL;
    xAutoExtend : BOOL;  // 自动伸出
	// 自动缩回
	xAutoRetract: BOOL;
    xReset : BOOL;  // 复位按钮
    xPosExtend : BOOL;  // 伸出到位传感器
    xPosRetract : BOOL;  // 缩回到位传感器
    tTimeout : TIME := T#5S;  // 动作超时时间
END_VAR
VAR_OUTPUT
    yValve1 : BOOL;  // 电磁阀1输出：TRUE=伸出，FALSE=缩回
	// 电磁阀2输出：TRUE=伸出，FALSE=缩回
	yValve2: BOOL;
    bAlarm : BOOL;  // 报警输出
END_VAR
VAR
    bEnableCmd1 : BOOL;  // 有效的命令1
	// 有效的命令1
	bEnableCmd2: BOOL;
	tActionTimer: TON;// 动作定时器
END_VAR
VAR_INPUT
	// 气缸类型  0 单控  1双控
	cylinder_type: INT;
END_VAR



CASE cylinder_type OF
	0:     //单控电池阀
		//命令逻辑选择
		IF xManualAuto  THEN
			//自动模式，使用自动命令
			bEnableCmd1 :=xAutoExtend;
			ELSE
			//手动模式，使用手动命令
			bEnableCmd1 :=xManualExtend  ;
		END_IF
		//控制指令
		IF bEnableCmd1 THEN
			//开始伸出
			yValve1:=TRUE;
			ELSE
			//开始缩回
			yValve1 :=FALSE;
		END_IF
		
	
			tActionTimer(IN := (NOT xPosExtend AND NOT yValve1)  OR   (NOT xPosRetract AND yValve1), PT:=tTimeout );
			bAlarm :=tActionTimer .Q;
	
	1:        //双控电池阀
		//命令逻辑选择
		IF xManualAuto  THEN
			//自动模式，使用自动命令
			bEnableCmd1 :=xAutoExtend;
			bEnableCmd2 :=xAutoRetract;
		ELSE
			//手动模式，使用手动命令
			bEnableCmd1 :=xManualExtend;
			bEnableCmd2 :=xManualRetract;
		END_IF
		//伸出控制指令
		IF bEnableCmd1 THEN
			//开始伸出
			yValve1:=TRUE;
			yValve2:=FALSE;
		ELSE 
			yValve1:=FALSE;
		END_IF
		
		IF bEnableCmd2 THEN
			//开始缩回
			yValve2:=TRUE;
			yValve1:=FALSE;
		ELSE 
			yValve2:=FALSE;
		END_IF
		
			tActionTimer(IN := (NOT xPosExtend AND NOT yValve1)  OR   (NOT xPosRetract AND yValve2), PT:=tTimeout );
			bAlarm :=tActionTimer .Q;
		
END_CASE

IF xReset THEN
	bAlarm:=FALSE ;
END_IF

END_FUNCTION_BLOCK

// Device/Application/40_Man/PLC_PCManual
PROGRAM PLC_PCManual
VAR
	// ══ PC 单点控制握手 (上位机 ManualService 读写; 其余 POU 只读 PC_Manual_Active) ══
	// pragma 不可省: 新对象默认不进符号配置, 漏写则 OPC UA browse 不到、上位机写入被静默丢弃。
	{attribute 'symbol' := 'readwrite'}
	PC_Manual_Enable: BOOL;        // PC→PLC: 请求进入单点模式 (电平; 退出写 FALSE)
	{attribute 'symbol' := 'readwrite'}
	PC_Manual_Keepalive: DINT;     // PC→PLC: 心跳, 上位机每秒 +1; 停变满 3s 判死 (只看变没变, 回绕安全)
	{attribute 'symbol' := 'read'}
	PC_Manual_Active: BOOL;        // PLC→PC: 单点模式实际生效 —— 唯一权威判定, 上位机据此才允许下发
	                               // 同时被 A00_设备状态显示及控制 消费: 为真即强制电子手动档
	{attribute 'symbol' := 'read'}
	PC_Manual_Reject: INT;         // PLC→PC: Enable 为真却未生效的原因
	                               // 0=无 1=心跳超时 2=L2占用 3=PLC未就绪 4=下载握手中

	iLastKeepalive: DINT;
	tonKeepalive: TON;
	bL2AllIdle: BOOL;
	bGateOk: BOOL;
	ftActive: F_TRIG;
END_VAR

// ════════════════════════════════════════════════════════════════════════════
// PC 单点控制 (PC Manual Mode) —— 上位机的"电子手动档"
//
// HMI 手动屏的按钮只在柜面手/自动旋钮打到"手动"时生效: FB_cylinder 里
// `IF xManualAuto THEN 用自动位 ELSE 用手动位`, 而 xManualAuto 接的就是 ManualAuto。
// 本 POU 算出的 PC_Manual_Active 被 A00_设备状态显示及控制 接进 FB_Mode 的 xAutoMode:
//     xAutoMode := 手自动 AND NOT PLC_PCManual.PC_Manual_Active
// 于是上位机一进单点, 整机就切到手动档 —— 等效于有人拧了旋钮, 机器不会进入任何
// 它没被设计过的状态。上位机因此**只写 <设备>手动 位** (与 HMI 手动屏同一批位),
// 完全不碰 <设备>自动 —— 那是 L2 流程与 PLC_Pump_泵管理 的地盘, 抢它必然打架。
//
// 顺带白捡两个结构性好处:
//   · FB_Mode 的 `ELSIF (bAuto AND xStart)` 决定手动档下「启动」不被接受 ——
//     单点会话激活期间机器根本无法被启动进运行态, 不必在软件里另设防线。
//   · 手轮用的是**原始物理输入** (bHandWheelAllowed := ... AND NOT 手自动),
//     电子手动档不会把手轮放出来, 这是有意为之。
//
// 伺服轴不受档位影响 (FB_SERVOAXIS 的 bNormalMotionAllowed 只看通信/使能/PLC_Ready),
// 故轴无需任何改造, 上位机直接写 <轴>DATE 的命令位。
//
// Active 为真的必要条件, 任一失守立即落下并清扫:
//   1. 上位机心跳 3s 内有跳变      —— 断网 / 后端崩溃 / 前端卡死自动收口
//   2. 8 个工位 L2 全部非 RUNNING  —— 与上位机自身的动作 / 流程互斥
//   3. PLC_Ready 且不在下载握手中  —— 与 PLC 全下载维护窗口互斥
// (不再要求 MODE_State<>运行: 既然不写自动位, L2 派发器与泵管理写什么都被 FB 忽略,
//  两个写者的问题不存在, 也就不必先把设备停下来。)
//
// Active 下降沿一次性清扫 51 个执行器的**手动位**与 11 根轴的运动命令位:
// OPC UA 写进去的是电平而非脉冲, 上位机若在阀通电时崩溃, 不清扫阀就会一直通着。
// 只清手动位: 自动位从头到尾没被我们碰过, 档位一还原, 各执行器自然接着听流程的。
// 不清 xStop (安全方向) 与 XReset (清错方向)。
// ════════════════════════════════════════════════════════════════════════════

// ── 1. 8 工位 L2 空闲 (10 = RUNNING) ──
bL2AllIdle := (Host_Computer.Sampling_L2_State <> 10)
	AND (Host_Computer.Collect_L2_State <> 10)
	AND (Host_Computer.Develop_L2_State <> 10)
	AND (Host_Computer.PhotoScrape_L2_State <> 10)
	AND (Host_Computer.FeedLift_L2_State <> 10)
	AND (Host_Computer.Pump_L2_State <> 10)
	AND (Host_Computer.Rail_L2_State <> 10)
	AND (Host_Computer.StagingA_L2_State <> 10);

// ── 2. 心跳看门狗: 值有跳变即复位计时 ──
IF PC_Manual_Keepalive <> iLastKeepalive THEN
	iLastKeepalive := PC_Manual_Keepalive;
	tonKeepalive(IN := FALSE, PT := T#3S);
END_IF
tonKeepalive(IN := PC_Manual_Enable, PT := T#3S);

// ── 3. 生效判定 ──
bGateOk := PLC_Ready AND ((PLC_Deploy_State = 0) OR (PLC_Deploy_State = 30));
PC_Manual_Active := PC_Manual_Enable AND NOT tonKeepalive.Q AND bL2AllIdle AND bGateOk;

// ── 4. 拒绝原因回显 (上位机面板直接显示"为什么点不动") ──
IF NOT PC_Manual_Enable THEN
	PC_Manual_Reject := 0;
ELSIF tonKeepalive.Q THEN
	PC_Manual_Reject := 1;
ELSIF NOT bL2AllIdle THEN
	PC_Manual_Reject := 2;
ELSIF NOT PLC_Ready THEN
	PC_Manual_Reject := 3;
ELSIF (PLC_Deploy_State <> 0) AND (PLC_Deploy_State <> 30) THEN
	PC_Manual_Reject := 4;
ELSE
	PC_Manual_Reject := 0;
END_IF

// ── 5. Active 下降沿: 清扫全部 PC 可写的执行器手动位 / 轴命令位 ──
ftActive(CLK := PC_Manual_Active);
IF ftActive.Q THEN
	// 展缸 1/2 各 4 气缸
	展缸1气缸1手动 := FALSE;
	展缸1气缸2手动 := FALSE;
	展缸1气缸3手动 := FALSE;
	展缸1气缸4手动 := FALSE;
	展缸2气缸1手动 := FALSE;
	展缸2气缸2手动 := FALSE;
	展缸2气缸3手动 := FALSE;
	展缸2气缸4手动 := FALSE;
	// 展缸 1 进液 / 排液 / 吹气电池阀
	展缸1进液电池阀1手动 := FALSE;
	展缸1进液电池阀2手动 := FALSE;
	展缸1进液电池阀3手动 := FALSE;
	展缸1进液电池阀4手动 := FALSE;
	展缸1排液电池阀1手动 := FALSE;
	展缸1排液电池阀2手动 := FALSE;
	展缸1排液电池阀3手动 := FALSE;
	展缸1排液电池阀4手动 := FALSE;
	展缸1吹气电池阀1手动 := FALSE;
	展缸1吹气电池阀2手动 := FALSE;
	展缸1吹气电池阀3手动 := FALSE;
	展缸1吹气电池阀4手动 := FALSE;
	// 展缸 2 进液 / 排液 / 吹气电池阀
	展缸2进液电池阀1手动 := FALSE;
	展缸2进液电池阀2手动 := FALSE;
	展缸2进液电池阀3手动 := FALSE;
	展缸2进液电池阀4手动 := FALSE;
	展缸2排液电池阀1手动 := FALSE;
	展缸2排液电池阀2手动 := FALSE;
	展缸2排液电池阀3手动 := FALSE;
	展缸2排液电池阀4手动 := FALSE;
	展缸2吹气电池阀1手动 := FALSE;
	展缸2吹气电池阀2手动 := FALSE;
	展缸2吹气电池阀3手动 := FALSE;
	展缸2吹气电池阀4手动 := FALSE;
	// 收集工位
	收集下压气缸手动 := FALSE;
	收集夹持气缸手动 := FALSE;
	收集升降气缸手动 := FALSE;
	收集伸缩气缸手动 := FALSE;
	收集进液手动 := FALSE;
	收集排液手动 := FALSE;
	收集正压排液手动 := FALSE;
	溶液收集瓶定位手动 := FALSE;
	// 拍照刮板工位
	刮板拍照遮光气缸手动 := FALSE;
	刮板拍照旋转气缸手动 := FALSE;
	刮板拍照下压气缸手动 := FALSE;
	刮板拍照真空手动 := FALSE;
	刮板拍照无刷电机手动 := FALSE;
	刮板拍照定位气缸手动 := FALSE;
	// 上样点样工位
	上样定位手动 := FALSE;
	上样点样三通电池阀手动 := FALSE;
	上样吹气手动 := FALSE;
	// 泵站 / 中转
	大真空泵手动 := FALSE;
	粉末收集器定位手动 := FALSE;

	// 11 根伺服轴的运动命令位 (不清 xStop / XReset)
	玻璃上料轴1ZDATE.xJogPos := FALSE; 玻璃上料轴1ZDATE.xJogNeg := FALSE;
	玻璃上料轴1ZDATE.xMoveAbs := FALSE; 玻璃上料轴1ZDATE.xMoveRel := FALSE; 玻璃上料轴1ZDATE.xHome := FALSE;
	玻璃上料轴2ZDATE.xJogPos := FALSE; 玻璃上料轴2ZDATE.xJogNeg := FALSE;
	玻璃上料轴2ZDATE.xMoveAbs := FALSE; 玻璃上料轴2ZDATE.xMoveRel := FALSE; 玻璃上料轴2ZDATE.xHome := FALSE;
	打样瓶上料轴3YDATE.xJogPos := FALSE; 打样瓶上料轴3YDATE.xJogNeg := FALSE;
	打样瓶上料轴3YDATE.xMoveAbs := FALSE; 打样瓶上料轴3YDATE.xMoveRel := FALSE; 打样瓶上料轴3YDATE.xHome := FALSE;
	上样轴4X轴DATE.xJogPos := FALSE; 上样轴4X轴DATE.xJogNeg := FALSE;
	上样轴4X轴DATE.xMoveAbs := FALSE; 上样轴4X轴DATE.xMoveRel := FALSE; 上样轴4X轴DATE.xHome := FALSE;
	上样轴5Z轴DATE.xJogPos := FALSE; 上样轴5Z轴DATE.xJogNeg := FALSE;
	上样轴5Z轴DATE.xMoveAbs := FALSE; 上样轴5Z轴DATE.xMoveRel := FALSE; 上样轴5Z轴DATE.xHome := FALSE;
	点样轴6XDATE.xJogPos := FALSE; 点样轴6XDATE.xJogNeg := FALSE;
	点样轴6XDATE.xMoveAbs := FALSE; 点样轴6XDATE.xMoveRel := FALSE; 点样轴6XDATE.xHome := FALSE;
	点样轴7YDATE.xJogPos := FALSE; 点样轴7YDATE.xJogNeg := FALSE;
	点样轴7YDATE.xMoveAbs := FALSE; 点样轴7YDATE.xMoveRel := FALSE; 点样轴7YDATE.xHome := FALSE;
	拍照轴8YDATE.xJogPos := FALSE; 拍照轴8YDATE.xJogNeg := FALSE;
	拍照轴8YDATE.xMoveAbs := FALSE; 拍照轴8YDATE.xMoveRel := FALSE; 拍照轴8YDATE.xHome := FALSE;
	刮板轴9XDATE.xJogPos := FALSE; 刮板轴9XDATE.xJogNeg := FALSE;
	刮板轴9XDATE.xMoveAbs := FALSE; 刮板轴9XDATE.xMoveRel := FALSE; 刮板轴9XDATE.xHome := FALSE;
	刮板轴10ZDATE.xJogPos := FALSE; 刮板轴10ZDATE.xJogNeg := FALSE;
	刮板轴10ZDATE.xMoveAbs := FALSE; 刮板轴10ZDATE.xMoveRel := FALSE; 刮板轴10ZDATE.xHome := FALSE;
	地轨轴11YDATE.xJogPos := FALSE; 地轨轴11YDATE.xJogNeg := FALSE;
	地轨轴11YDATE.xMoveAbs := FALSE; 地轨轴11YDATE.xMoveRel := FALSE; 地轨轴11YDATE.xHome := FALSE;
END_IF

END_PROGRAM

// Device/Application/25_FB_功能块/FB_Mode
FUNCTION_BLOCK FB_Mode
VAR_INPUT
    xStart      : BOOL;  // 启动按钮
    xStop       : BOOL;  // 停止按钮
    xReset      : BOOL;  // 复位按钮
    xAutoMode   : BOOL;  // TRUE=自动模式，FALSE=手动模式
    xFault      : BOOL;  // 故障信号
    xEmergency  : BOOL;  // 急停信号（急停按下为FALSE）
END_VAR
VAR_OUTPUT
    bRed        : BOOL;  // 红灯
    bYellow     : BOOL;  // 黄灯
    bGreen      : BOOL;  // 绿灯
    bBuzzer     : BOOL;  // 蜂鸣器
    iState      : INT;   // 设备状态: 0=停止, 1=运行, 2=故障, 3=急停
    bAuto       : BOOL;  // 自动模式指示
END_VAR
VAR
    iDeviceState : INT := 0;  // 0=停止, 1=运行, 2=故障, 3=急停
    
    // 定时器
    tBuzzerPulse : TON;  // 蜂鸣器脉冲
    tFlashTimer  : TON;  // 闪烁定时器
    tShortBeep   : TON;  // 短鸣定时器
    tEmergencyBeep : TON; // 急停蜂鸣器定时器
	// 蜂鸣器激活
	tEmergencyBeep1: TON;
    
    // 标志
    bBuzzerActive : BOOL := FALSE;  // 蜂鸣器激活
    bFlashFlag    : BOOL;           // 闪烁标志
    bBeepOnce     : BOOL := FALSE;  // 单次蜂鸣标志
    bEmergencyBuzzer : BOOL := FALSE; // 急停蜂鸣器标志
    bEmergencyActive : BOOL := FALSE; // 急停激活标志
	ALT_0: ALT;
	ALT_1: ALT;
	TON_0: TON;
	ALT_2: ALT;
	TON_1: TON;
	TON_2: TON;
END_VAR
VAR_INPUT
	bWarning_alarm: BOOL;
END_VAR

// 模式状态
bAuto := xAutoMode;

// 状态机
CASE iDeviceState OF
    EN_功能块状态.停止:  // 停止状态
        IF NOT xEmergency THEN
            iDeviceState := EN_功能块状态.急停;  // 急停
            bEmergencyActive := TRUE;
        ELSIF xFault THEN
            iDeviceState := EN_功能块状态.故障;  // 故障
            bBuzzerActive := TRUE;
        ELSIF (bAuto AND xStart)  THEN
		 bBeepOnce := TRUE;  // 启动短鸣
		  iDeviceState := EN_功能块状态.初始化;  // 初始化

        END_IF;
    
    EN_功能块状态.运行:  // 运行状态
        IF NOT xEmergency THEN
            iDeviceState := EN_功能块状态.急停;  // 急停
            bEmergencyActive := TRUE;
        ELSIF xFault THEN
            iDeviceState := EN_功能块状态.故障;  // 故障
            bBuzzerActive := TRUE;
        ELSIF xStop THEN
            iDeviceState := EN_功能块状态.停止;  // 停止
            bBeepOnce := TRUE;  // 停止短鸣
        END_IF;
        
    EN_功能块状态.故障:  // 故障状态
        IF NOT xEmergency THEN
            iDeviceState := EN_功能块状态.急停;  // 急停
            bEmergencyActive := TRUE;
        ELSIF xReset AND NOT xFault THEN
            iDeviceState := EN_功能块状态.停止;  // 停止
            bBuzzerActive := FALSE;
			bBuzzer:=FALSE;
        END_IF;
        
    EN_功能块状态.急停:  // 急停状态
        // 急停复位需要：急停信号解除 + 复位按钮按下
        IF  xEmergency AND xReset THEN
            iDeviceState := EN_功能块状态.停止;  // 停止
            bEmergencyActive := FALSE;
            bEmergencyBuzzer := FALSE;
			bBuzzer:=FALSE;
        END_IF;
	EN_功能块状态.初始化:  //初始化状态
	 TON_0(IN:=TRUE , PT:=T#3S );
		IF TON_0.Q THEN
		iDeviceState := EN_功能块状态.运行;  // 运行
		END_IF 
END_CASE;

// 急停蜂鸣器控制（急停时蜂鸣器以不同频率鸣响）
IF  bEmergencyActive THEN
    tEmergencyBeep(IN := NOT tEmergencyBeep.Q, PT := T#2S );
	ALT_1(xExecute:= tEmergencyBeep.Q, xOut:=bBuzzer );  // 急停时蜂鸣器响2秒，停2秒	
END_IF;

//三色灯控制
// 闪烁定时器
tFlashTimer(IN := NOT tFlashTimer.Q, PT := T#500MS);
ALT_0(xExecute:=tFlashTimer.Q , xOut:=bFlashFlag );

CASE iDeviceState OF
    EN_功能块状态.停止:  // 停止状态
        IF bAuto THEN
            bYellow := TRUE;           // 自动模式：黄灯常亮
        ELSE
            bYellow := bFlashFlag;     // 手动模式：黄灯闪烁
        END_IF;
		 bGreen :=FALSE;
		 bRed :=FALSE;
        
    EN_功能块状态.运行:  // 运行状态
        bGreen := TRUE;
         bRed :=FALSE;
		  bYellow := FALSE; 
    EN_功能块状态.故障:  // 故障状态
        bRed := TRUE;
         bGreen :=FALSE;
		 bYellow := FALSE; 
    EN_功能块状态.急停:  // 急停状态
        bRed := bFlashFlag;  // 红灯闪烁
		bGreen :=FALSE;
		 bYellow := FALSE; 
END_CASE;
tShortBeep(IN := bBeepOnce AND NOT bEmergencyActive, PT := T#500MS);
// 蜂鸣器控制
IF bBeepOnce AND NOT bEmergencyActive THEN
	bBuzzer := TRUE;  // 短鸣
    IF tShortBeep.Q THEN
        bBeepOnce := FALSE;
       bBuzzer := FALSE;
    END_IF;
    
END_IF;

// 故障时蜂鸣器（非急停状态时生效）
IF NOT bEmergencyActive AND xFault  THEN
    tBuzzerPulse(IN := NOT tBuzzerPulse.Q, PT := T#500MS);
ALT_2(xExecute:= tBuzzerPulse.Q, xOut:= bBuzzer);
END_IF;


//蜂鸣器5S后停止
TON_2(IN:=iDeviceState=2 OR iDeviceState=3 OR bWarning_alarm ,PT:=T#5S);
IF TON_2.Q THEN
	bBuzzer:=FALSE;
END_IF

IF bWarning_alarm AND NOT TON_2.Q THEN
	bBuzzer:=TRUE;
	
END_IF
IF bWarning_alarm  THEN
	 bRed := TRUE;
	  
END_IF

IF xReset THEN
	bBuzzer:=FALSE;
	bRed := FALSE;
END_IF



// 输出状态
iState := iDeviceState;

END_FUNCTION_BLOCK

// Device/Application/50_action/PLC_Pump_泵管理
PROGRAM PLC_Pump_泵管理
VAR
	bPumpCommandsArmed: BOOL;
	bAnyPumpCommandRequested: BOOL;

END_VAR

// PLC deploy vacuum gate
(* 真空泵集中管理: 大真空泵站位[] 引用计数总线 -> 大真空泵自动
   -> FB_cylinder cylinder_8 -> 大真空泵 %QX2.4。State30 是忙拒绝，已有真空继续；
   启动/维护期间写入的站位必须全部回 FALSE 后才重新装载，禁止解锁时补执行。 *)
bAnyPumpCommandRequested := 大真空泵站位[0]
	OR 大真空泵站位[1]
	OR 大真空泵站位[2]
	OR 大真空泵站位[3]
	OR 大真空泵站位[4]
	OR 大真空泵站位[5]
	OR 大真空泵站位[6]
	OR 大真空泵站位[7]
	OR 大真空泵站位[8]
	OR 大真空泵站位[9]
	OR 大真空泵站位[10]
	OR 大真空泵站位[11];
IF ((NOT PLC_Ready) OR ((PLC_Deploy_State<>0) AND (PLC_Deploy_State<>30))) THEN
	bPumpCommandsArmed := FALSE;
ELSIF NOT bAnyPumpCommandRequested THEN
	bPumpCommandsArmed := TRUE;
END_IF
大真空泵自动 := PLC_Ready AND ((PLC_Deploy_State=0) OR (PLC_Deploy_State=30)) AND bPumpCommandsArmed AND bAnyPumpCommandRequested;

(* 上位机可观测性镜像 -> Host_Computer (只读诊断; 本 POU 每扫描运行, 借道镜像.
   Pump_Vacuum_On 是站位聚合+使能门后的泵命令态, 非接触器/真空度物理反馈;
   废液传感器 TRUE=该组废液管已走空, A26/排液判据共用此电平. *)
Pump_Vacuum_On := 大真空泵自动;
Expand_Waste_Empty_G1 := 展缸1溶剂废液检测传感器;
Expand_Waste_Empty_G2 := 展缸2溶剂废液检测传感器;

END_PROGRAM

// Device/Application/25_FB_功能块/FB_SERVOAXIS
FUNCTION_BLOCK FB_SERVOAXIS
VAR_IN_OUT
	AXIS: AXIS_REF_SM3;
END_VAR
VAR_INPUT
	xEnable    : BOOL;
	xStartupMotionAllowed : BOOL;       // TRUE only for the one axis owned by the startup homing FSM
	xHome      : BOOL;
	xJogPos    : BOOL;
	xJogNeg    : BOOL;
	xStop      : BOOL;
	xMoveAbs   : BOOL;
	xMoveRel   : BOOL;
	XReset     : BOOL;
	fAbsTarget : LREAL := 0.0;
	fRelTarget : LREAL := 0.0;
	fVelocity  : LREAL := 100.0;
	fAcc       : LREAL := 1000.0;
	fDec       : LREAL := 1000.0;
	fJogVel    : LREAL := 50.0;
END_VAR
VAR_OUTPUT
	bEnabled    : BOOL;
	bHomed      : BOOL;
	bBusy       : BOOL;
	bMotionBusy : BOOL;                 // motion-command busy only; excludes MC_Power.Busy (constant TRUE while enabled on Inovance SM3)
	bError      : BOOL;
	iErrorCode  : DINT;
	iFaultSource : INT;                 // 0 none,1 axis,2 power,3 home,4 abs,5 rel,6 halt,7 jog,8 reset,9 comm
	bCommOperational : BOOL;
	fActPos     : LREAL;
	fActVel     : LREAL;
	bAbMoveDone : BOOL;
	bReMoveDone : BOOL;
END_VAR
VAR
	MC_Power : MC_Power;
	MC_Home : MC_Home;
	MC_Halt : MC_Halt;
	MC_MoveAbsolute : MC_MoveAbsolute;
	MC_MoveRelative : MC_MoveRelative;
	MC_Jog : MC_Jog;
	MC_Reset : MC_Reset;
	CheckCommunication : SMC_CheckAxisCommunication;
	ResetAxisEdge : R_TRIG;
	ClearFaultEdge : R_TRIG;
	bPowerAllowed : BOOL;
	bNormalMotionAllowed : BOOL;
	bStartupMotionAllowed : BOOL;
	bFaultLatched : BOOL;
	iLatchedSource : INT;
	diLatchedCode : DINT;
END_VAR

// Always execute the communication diagnostic and all PLCopen FB instances cyclically.
CheckCommunication(Axis := AXIS, bEnable := TRUE);
bCommOperational := CheckCommunication.bValid AND CheckCommunication.bOperational;

// Power is allowed only after the startup FSM reached POWER and never while a download is prepared.
bPowerAllowed := bCommOperational
	AND (PLC_Startup_State >= 30) AND (PLC_Startup_State <> 90)
	AND ((PLC_Deploy_State = 0) OR (PLC_Deploy_State = 30));
bNormalMotionAllowed := bCommOperational AND bEnabled AND PLC_Ready
	AND ((PLC_Deploy_State = 0) OR (PLC_Deploy_State = 30));
bStartupMotionAllowed := bCommOperational AND bEnabled AND xStartupMotionAllowed
	AND (PLC_Startup_State >= 40) AND (PLC_Startup_State <= 51)
	AND ((PLC_Deploy_State = 0) OR (PLC_Deploy_State = 30));

// MC_Power 必须每扫描执行: PLCopen FB 在 Enable=FALSE 时不活动, 输出冻结在上次值 ——
// 若用 bPowerAllowed 驱动 Enable, 下载准备期 (PLC_Deploy_State=10) 的 Status 会一直保持
// 上一次的 TRUE, 使部署握手"等待全部去使能"永不成立 (实测 11 轴 bEnabled 全程 TRUE 到 10s
// 超时报 ErrorCode 40, 且驱动器实际从未断电)。故 Enable 只跟通信有效性, 真正的上下电由
// bRegulatorOn/bDriveStart 承载, Status 才能如实反映功率级状态。
MC_Power(
	Axis := AXIS,
	Enable := bCommOperational,
	bRegulatorOn := xEnable AND bPowerAllowed,
	bDriveStart := xEnable AND bPowerAllowed,
	Status => bEnabled);

MC_Home(
	Axis := AXIS,
	Execute := xHome AND (bNormalMotionAllowed OR bStartupMotionAllowed),
	Done => bHomed);

// MC_Reset is edge-triggered and is issued only for a communicating ErrorStop axis.
ResetAxisEdge(CLK := XReset AND bCommOperational AND (AXIS.nAxisState = 1));
ClearFaultEdge(CLK := XReset AND bCommOperational AND (AXIS.nAxisState <> 1));
MC_Reset(Axis := AXIS, Execute := ResetAxisEdge.Q);

MC_Jog(
	Axis := AXIS,
	JogForward := xJogPos AND bNormalMotionAllowed,
	JogBackward := xJogNeg AND bNormalMotionAllowed,
	Velocity := fJogVel,
	Acceleration := fAcc,
	Deceleration := fDec);

// Halt remains available whenever axis communication is valid.
MC_Halt(
	Axis := AXIS,
	Execute := xStop AND bCommOperational,
	Deceleration := fDec);

MC_MoveAbsolute(
	Axis := AXIS,
	Execute := xMoveAbs AND bNormalMotionAllowed,
	Position := fAbsTarget,
	Velocity := fVelocity,
	Acceleration := fAcc,
	Deceleration := fDec,
	Done => bAbMoveDone);

MC_MoveRelative(
	Axis := AXIS,
	Execute := xMoveRel AND (bNormalMotionAllowed OR bStartupMotionAllowed),
	Distance := fRelTarget,
	Velocity := fVelocity,
	Acceleration := fAcc,
	Deceleration := fDec,
	Done => bReMoveDone);

fActPos := AXIS.fActPosition;
fActVel := AXIS.fActVelocity;
bBusy := MC_Power.Busy OR MC_Home.Busy OR MC_Halt.Busy OR MC_MoveAbsolute.Busy
	OR MC_MoveRelative.Busy OR MC_Jog.Busy OR MC_Reset.Busy;
// 运动忙 (不含 MC_Power.Busy): 汇川 SM3 的 MC_Power 使能期间 Busy 恒为 TRUE, 混入会使部署门禁在就绪态永久误报
bMotionBusy := MC_Home.Busy OR MC_Halt.Busy OR MC_MoveAbsolute.Busy
	OR MC_MoveRelative.Busy OR MC_Jog.Busy OR MC_Reset.Busy;

// Preserve the first real motion/drive fault. Communication loss is reported separately and never
// fanned out as eleven servo faults. Axis state 2 is Stopping and is deliberately not an error.
IF (MC_Reset.Done AND (AXIS.nAxisState <> 1)) OR ClearFaultEdge.Q THEN
	bFaultLatched := FALSE;
	iLatchedSource := 0;
	diLatchedCode := 0;
ELSIF NOT bFaultLatched AND bCommOperational THEN
	IF MC_Power.Error THEN
		bFaultLatched := TRUE; iLatchedSource := 2; diLatchedCode := MC_Power.ErrorID;
	ELSIF MC_Home.Error THEN
		bFaultLatched := TRUE; iLatchedSource := 3; diLatchedCode := MC_Home.ErrorID;
	ELSIF MC_MoveAbsolute.Error THEN
		bFaultLatched := TRUE; iLatchedSource := 4; diLatchedCode := MC_MoveAbsolute.ErrorID;
	ELSIF MC_MoveRelative.Error THEN
		bFaultLatched := TRUE; iLatchedSource := 5; diLatchedCode := MC_MoveRelative.ErrorID;
	ELSIF MC_Halt.Error THEN
		bFaultLatched := TRUE; iLatchedSource := 6; diLatchedCode := MC_Halt.ErrorID;
	ELSIF MC_Jog.Error THEN
		bFaultLatched := TRUE; iLatchedSource := 7; diLatchedCode := MC_Jog.ErrorID;
	ELSIF MC_Reset.Error THEN
		bFaultLatched := TRUE; iLatchedSource := 8; diLatchedCode := MC_Reset.ErrorID;
	ELSIF AXIS.nAxisState = 1 THEN
		bFaultLatched := TRUE;
		iLatchedSource := 1;
		// Prefer the drive's original diagnostic value; keep 1 only as an explicit unknown fallback.
		diLatchedCode := AXIS.diDriverErrorCode;
		IF diLatchedCode = 0 THEN diLatchedCode := 1; END_IF
	END_IF
END_IF

bError := bFaultLatched;
IF NOT bCommOperational THEN
	iFaultSource := 9;
	iErrorCode := WORD_TO_DINT(CheckCommunication.wComState);
ELSE
	iFaultSource := iLatchedSource;
	iErrorCode := diLatchedCode;
END_IF

END_FUNCTION_BLOCK

// Device/Application/50_action/Rail_Sync
PROGRAM Rail_Sync
VAR
	i : INT;
END_VAR

(* 地轨 11Y 双源同步桥 (非动作派发器, 是 PC<->HMI 点位对账工具).
   原理: HMI_地轨轴11Y.position[] 是单 ExtensionObject struct, OPC 逐成员读写不可行
         -> 让 PLC 当桥, OPC 只暴露 flat 数组 (复用 *_ActPos 镜像同套路).
   每扫描无条件执行 (挂 PLC_MainPRG 无条件段, 与 ActPos 镜像同处; 勿放运行态 CASE).
   守恒: PUSH 纯 PLC 内存拷贝, 任一侧可触发; PULL 写真源恒为 PC, HMI 触发=请 PC 提交. *)

// (1) 常开镜像: HMI 教值 -> flat 只读镜像 (PC 经此读做 diff/pull, 不直访 struct)
FOR i := 1 TO 6 DO
	Rail_Pos_HMI[i] := HMI_地轨轴11Y.position[i];
END_FOR

// (2) 同步邮箱
CASE Rail_Sync_Req OF
	1:  (* PUSH: PC 真源 Rail_Pos_Target[] -> HMI 工作副本 position[] (PLC 写自己 struct, 无 OPC 限制) *)
		FOR i := 1 TO 6 DO
			HMI_地轨轴11Y.position[i] := Rail_Pos_Target[i];
		END_FOR
		Rail_Sync_Ack := 1;     (* 完成 *)
		Rail_Sync_Req := 0;     (* 清请求 *)

	2:  (* PULL: 收现场教值回真源. PLC 写不了 yaml, 更不可碰 Rail_Pos_Target (单写者=PC).
	          -> 仅亮邮箱待 PC 提交. PC 轮询见 Req=2 -> 读 Rail_Pos_HMI[] -> 限位校验/diff/确认
	             -> 写 points.yaml + 重算并写 Rail_Pos_Target[] -> 由 PC 置 Req:=0,Ack:=1 (失败 Ack:=3). *)
		Rail_Sync_Ack := 2;     (* 待 PC 提交 (PC 接手后由 PC 改写 Ack/Req) *)
END_CASE

END_PROGRAM

// Device/Application/30_Ethercat任务/PLC_CNC
PROGRAM PLC_CNC
VAR
	SMC_Interpolator: SMC_Interpolator;
	SMC_ControlAxisByPos1: SMC_ControlAxisByPos;
	SMC_ControlAxisByPos2: SMC_ControlAxisByPos;
	SMC_ControlAxisByPos3: SMC_ControlAxisByPos;
	SMC_TRAFO_Gantry3: SMC_TRAFO_Gantry3;
	SMC_TRAFOF_Gantry3: SMC_TRAFOF_Gantry3;
	SMC_NCDecoder_0: SMC_NCDecoder;
	SMC_CheckVelocities: SMC_CheckVelocities;
	SMC_SmoothPath: SMC_SmoothPath;
	SR: SR;
	RS: RS;
END_VAR
VAR // added by the converter: edge detectors and wires of the graphical bodies
    _w1, _w2, _w3 : BOOL;
    _w4, _w5 : ANY;
END_VAR

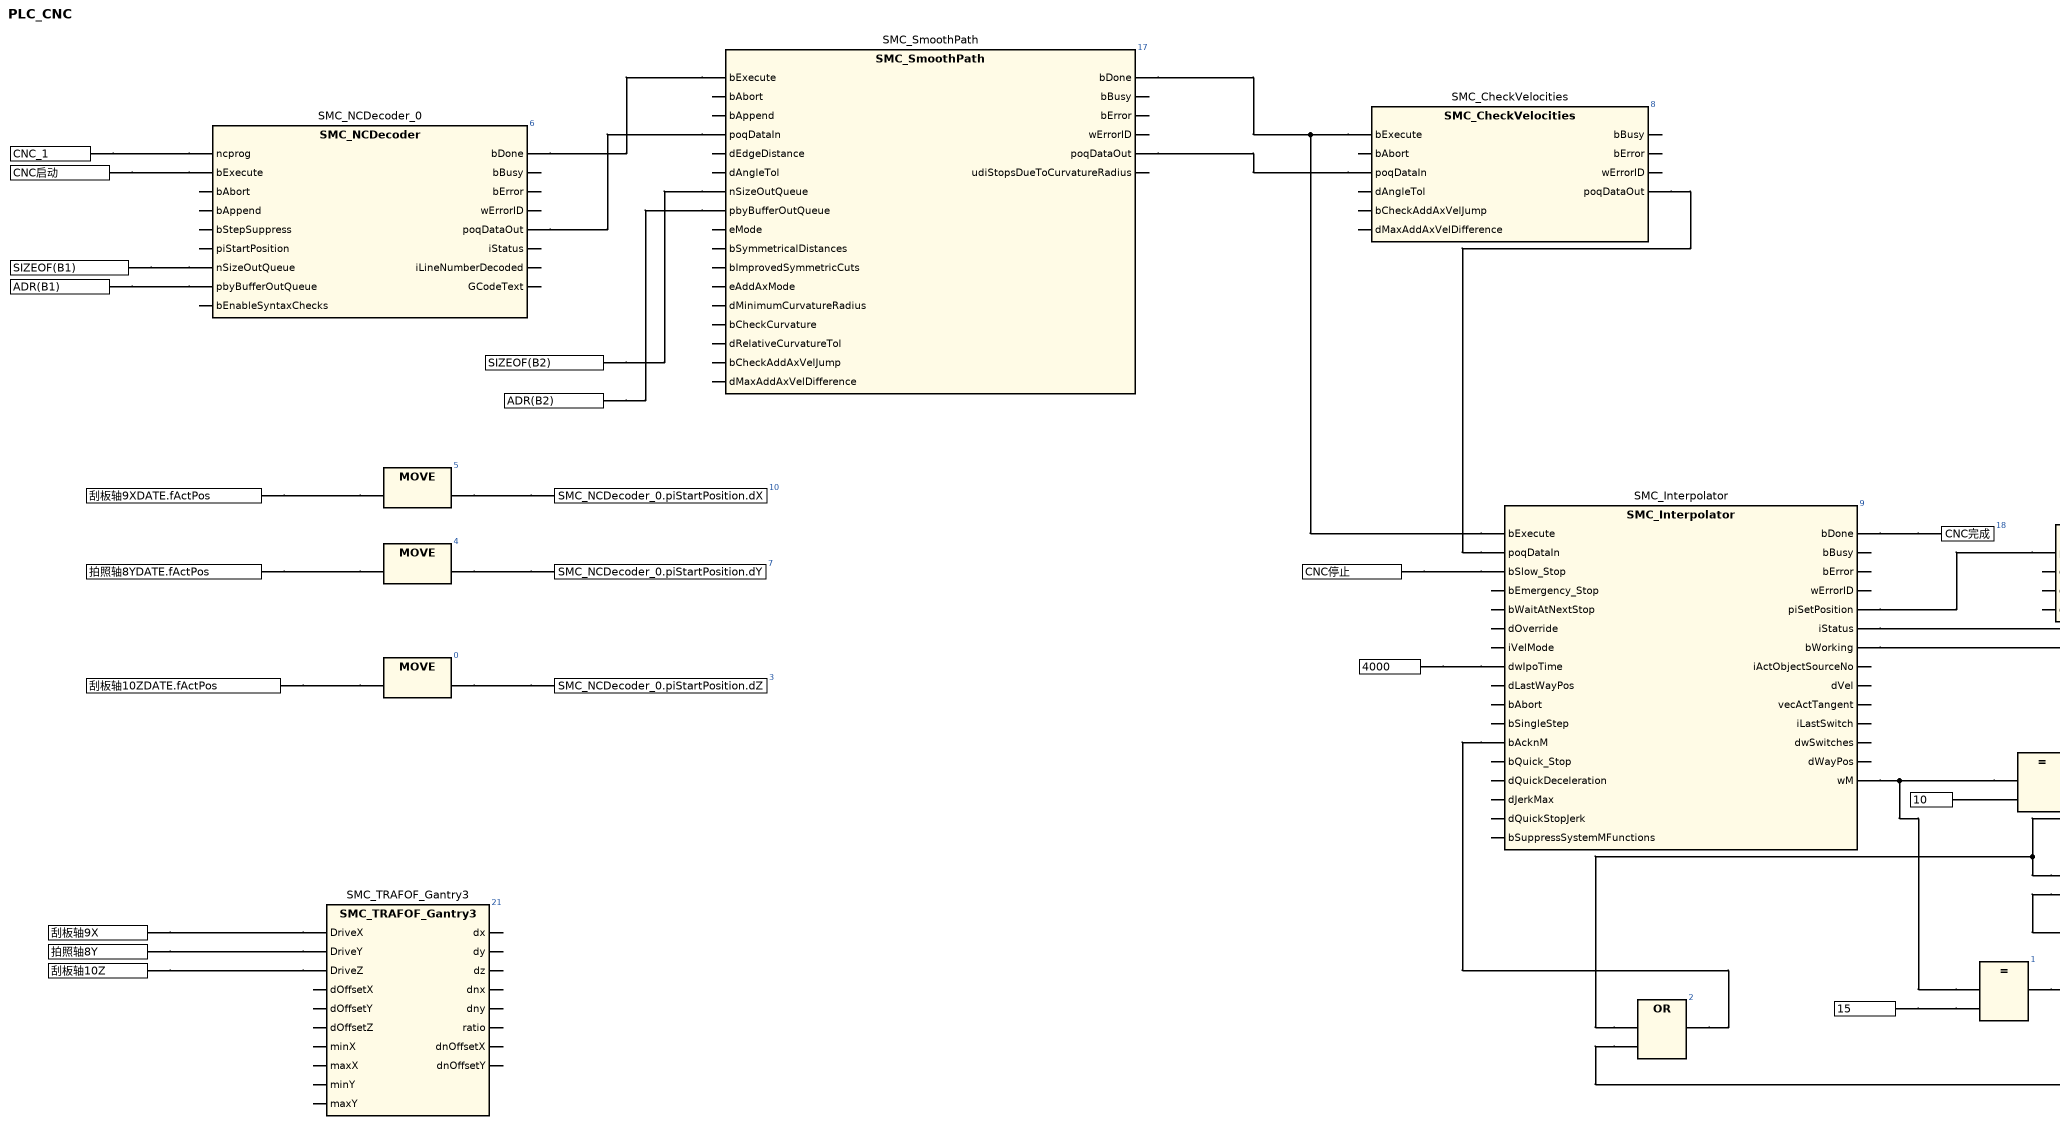
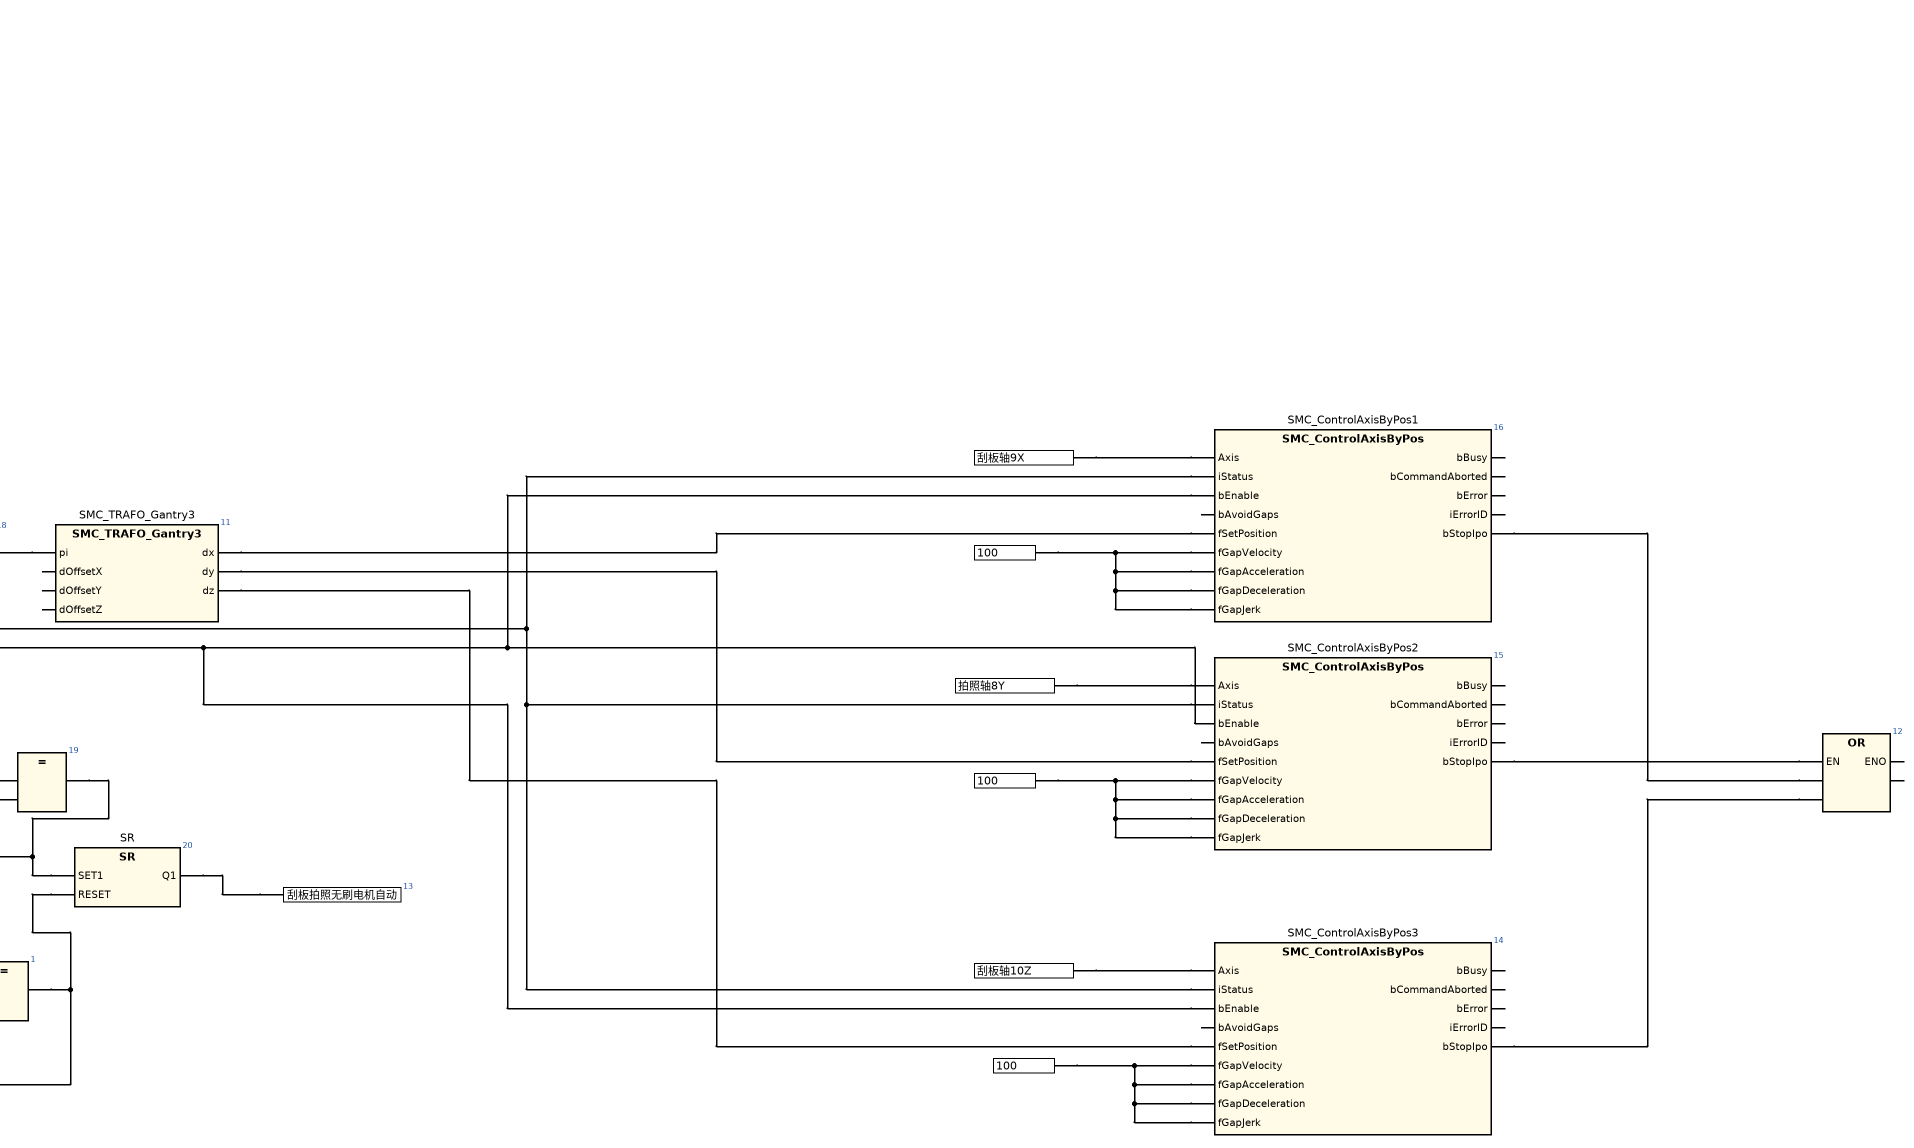
// note: 4 stored wires end on pins the file does not list and are not shown
_w1 := SMC_Interpolator.wM = 15;
_w3 := _w2 OR _w1;
SMC_NCDecoder_0.piStartPosition.dZ := 刮板轴10ZDATE.fActPos;
_w4 := 拍照轴8YDATE.fActPos;
_w5 := 刮板轴9XDATE.fActPos;
SMC_NCDecoder_0(
    ncprog := CNC_1,
    bExecute := CNC启动,
    nSizeOutQueue := SIZEOF(B1),
    pbyBufferOutQueue := ADR(B1)); // SMC_NCDecoder
SMC_NCDecoder_0.piStartPosition.dY := _w4;
SMC_CheckVelocities(bExecute := SMC_SmoothPath.bDone, poqDataIn := SMC_SmoothPath.poqDataOut);
SMC_Interpolator(
    bExecute := SMC_SmoothPath.bDone,
    poqDataIn := SMC_CheckVelocities.poqDataOut,
    bSlow_Stop := CNC停止,
    dwIpoTime := 4000,
    bAcknM := _w3);
SMC_NCDecoder_0.piStartPosition.dX := _w5;
SMC_TRAFO_Gantry3(pi := SMC_Interpolator.piSetPosition);
IF SMC_ControlAxisByPos2.bStopIpo THEN (* SMC_ControlAxisByPos1.bStopIpo OR SMC_ControlAxisByPos3.bStopIpo; result not used *) END_IF
刮板拍照无刷电机自动 := SR.Q1;
SMC_ControlAxisByPos3(
    Axis := 刮板轴10Z,
    iStatus := SMC_Interpolator.iStatus,
    bEnable := SMC_Interpolator.bWorking,
    fSetPosition := SMC_TRAFO_Gantry3.dz,
    fGapVelocity := 100,
    fGapAcceleration := 100,
    fGapDeceleration := 100,
    fGapJerk := 100); // SMC_ControlAxisByPos
SMC_ControlAxisByPos2(
    Axis := 拍照轴8Y,
    iStatus := SMC_Interpolator.iStatus,
    bEnable := SMC_Interpolator.bWorking,
    fSetPosition := SMC_TRAFO_Gantry3.dy,
    fGapVelocity := 100,
    fGapAcceleration := 100,
    fGapDeceleration := 100,
    fGapJerk := 100); // SMC_ControlAxisByPos
SMC_ControlAxisByPos1(
    Axis := 刮板轴9X,
    iStatus := SMC_Interpolator.iStatus,
    bEnable := SMC_Interpolator.bWorking,
    fSetPosition := SMC_TRAFO_Gantry3.dx,
    fGapVelocity := 100,
    fGapAcceleration := 100,
    fGapDeceleration := 100,
    fGapJerk := 100); // SMC_ControlAxisByPos
SMC_SmoothPath(
    bExecute := SMC_NCDecoder_0.bDone,
    poqDataIn := SMC_NCDecoder_0.poqDataOut,
    nSizeOutQueue := SIZEOF(B2),
    pbyBufferOutQueue := ADR(B2));
CNC完成 := SMC_Interpolator.bDone;
_w2 := SMC_Interpolator.wM = 10;
SR(SET1 := _w2, RESET := _w1);
SMC_TRAFOF_Gantry3(DriveX := 刮板轴9X, DriveY := 拍照轴8Y, DriveZ := 刮板轴10Z);

END_PROGRAM

// Device/Application/50_action/PhotoScrape_L2
PROGRAM PhotoScrape_L2
VAR
	初始化step: INT;
	拍照step: INT;
	刮板收集step: INT;
	// ── 对位检查 42/43/44 内部状态 (spec 2026-07-16-photoscrape-align-check; worklog docs/superpowers/plans/2026-07-16-align-plc-worklog.md) ──
	alignstep: INT;
	align_tx: LREAL;              // 42: TargetX 帧变换后的 9X 轴坐标目标
	align_ty: LREAL;              // 42: TargetY 帧变换后的 8Y 轴坐标目标
	align_sav_vel_9X: LREAL;      // 42: 移动前暂存 RETAIN PERSISTENT 的 DATE.fVelocity, Done 恢复
	align_sav_vel_8Y: LREAL;
	align_sav_vel_10Z: LREAL;     // 44: 同上
	bActionDone: BOOL;
	bActionError: BOOL;
	L2_StartTrig: R_TRIG;
END_VAR
VAR CONSTANT
	// ── 对位检查守卫常量 (42/44; worklog Q5/Q6) ──
	// Z 高门: 与 伺服调用 里 9X/8Y 互锁 "刮板轴10ZDATE.fActPos<6" 同值同哲学; 一切 XY 移动只在 10Z 顶部
	ALIGN_Z_XY_GATE   : LREAL := 6.0;
	// Z 检查高度上限 = plate_surface_z_mm(20.5) - align_clearance_mm(2.5); 恒 < 20.5 永不触板面 (上机核对)
	ALIGN_Z_CHECK_MAX : LREAL := 18.0;
	// ⚠️ 板区 XY 软限位窗 (轴坐标 mm) — 占位: 上机 jog 到板四角读 9X/8Y ActPos 实测 ±5mm 后回填;
	// 勿照抄 host plate_origin (host frame 与轴 frame 疑似不同, worklog Q5 坐标系警示)。
	// 回填前 MIN>MAX = 空集 → 42 与 44(降) 恒拒动 ErrorCode 422/424 (安全默认)
	ALIGN_X_WIN_MIN   : LREAL := 0.0;
	ALIGN_X_WIN_MAX   : LREAL := -1.0;
	ALIGN_Y_WIN_MIN   : LREAL := 0.0;
	ALIGN_Y_WIN_MAX   : LREAL := -1.0;
	// ⚠️ 帧变换占位 (Target 与 g_sx/g_sy 同帧 → 轴坐标): axis = K*Target + O;
	// 上机核实 CNC 帧 = 轴帧则保持恒等(K=1,O=0), 否则实测回填 (worklog C2)
	ALIGN_FRAME_KX    : LREAL := 1.0;
	ALIGN_FRAME_OX    : LREAL := 0.0;
	ALIGN_FRAME_KY    : LREAL := 1.0;
	ALIGN_FRAME_OY    : LREAL := 0.0;
	// 显式保守速度 (mm/s): ST 无既有 MoveAbsolute 典型值(速度在持久 DATE.fVelocity), 42/44 必须显式设 (worklog C4/Q6); 上机试定
	ALIGN_VEL_XY      : LREAL := 40.0;
	ALIGN_VEL_Z       : LREAL := 5.0;   // 对齐既有唯一速度字面量 5.0 (伺服一键回原点退避)
END_VAR

(* PhotoScrape 工位 L2 统一动作派发器
   按 PhotoScrape_L2_ActionCode 派发到纯设备原子动作 (不含机器人/相机/CNC 握手).
   Start 上升沿接受请求 -> RUNNING 每周期调用对应原子 -> bActionDone=DONE / bActionError=ERROR. *)
L2_StartTrig(CLK := PhotoScrape_L2_Start);

(* Global deployment/startup gate: reject before any physical action is dispatched. *)
IF L2_StartTrig.Q AND (PhotoScrape_L2_State=0)
	AND ((NOT PLC_Ready) OR (PLC_Deploy_State<>0)) THEN
	PhotoScrape_L2_AcceptedSeq := PhotoScrape_L2_RequestSeq;
	PhotoScrape_L2_ActiveCode := PhotoScrape_L2_ActionCode;
	PhotoScrape_L2_ErrorCode := 190;
	PhotoScrape_L2_Retryable := TRUE;
	PhotoScrape_L2_CompletedSeq := PhotoScrape_L2_RequestSeq;
	PhotoScrape_L2_State := 30;
	RETURN;
END_IF

CASE PhotoScrape_L2_State OF
	0:  (* IDLE *)
		PhotoScrape_L2_Step := 0;
		IF L2_StartTrig.Q THEN
			PhotoScrape_L2_AcceptedSeq := PhotoScrape_L2_RequestSeq;
			PhotoScrape_L2_ActiveCode  := PhotoScrape_L2_ActionCode;
			PhotoScrape_L2_ErrorCode   := 0;
			PhotoScrape_L2_Retryable   := FALSE;
			bActionDone  := FALSE;
			bActionError := FALSE;
			初始化step := 0;
			拍照step := 0;
			刮板收集step := 0;
			alignstep := 0;
			(* 新动作被受理 = 解除上一次中止留下的 CNC 刹车 (闩锁与 CNC停止 的写者在 PLC_MainPRG 闸门块).
			   不在此直接写 CNC停止: 单写者纪律 —— MainPRG 闸门块每扫描在本 POU 之前运行, 双写会互相覆盖。 *)
			CNC_AbortLatch := FALSE;
			CASE PhotoScrape_L2_ActionCode OF
				10, 31, 32, 33, 34, 35, 36, 40, 41, 42, 43, 44, 51, 52:
					PhotoScrape_L2_SafeState := 0;
					PhotoScrape_L2_State     := 10;   (* RUNNING *)
			ELSE
				PhotoScrape_L2_ErrorCode    := 101;  (* 未知动作码 *)
				PhotoScrape_L2_Retryable    := TRUE;
				PhotoScrape_L2_CompletedSeq := PhotoScrape_L2_AcceptedSeq;
				PhotoScrape_L2_State        := 30;   (* REJECTED *)
			END_CASE
		END_IF

	10: (* RUNNING *)
		(* RUNNING 中 RESET: 中止挂死动作。CNC 的熄火由 PLC_MainPRG 闸门块据同一个
		   PhotoScrape_L2_Reset 置 CNC_AbortLatch 完成 (刹车须挂到下次受理, 不能只亮一扫描)。 *)
		IF PhotoScrape_L2_Reset THEN PhotoScrape_L2_State := 0; RETURN; END_IF
		CASE PhotoScrape_L2_ActiveCode OF
			10: A10_init_初始化();
			31: A31_cam_移轴335();
			32: A32_cam_定位();
			33: A33_cam_下压();
			36: 粉末收集器定位自动:=PhotoScrape_PowderCollectorLocate_Target; bActionDone:=TRUE;
			34: A34_cam_相机位();
			35: A35_cam_回零();
			40: A40_scrape_刮取();
			41: A41_scrape_收尾();
			51: A51_取料松压();
			52: A52_取料停旋转();

			(* ── 对位检查 42/43/44 (spec 2026-07-16-photoscrape-align-check §4; worklog 2026-07-16-align-plc-worklog.md)
			   内联原子 (codesys-mcp 无法新建 action POU); 专动作专用: 不碰 g_数组/收集器轴/气缸/真空/翻料 ── *)
			42: (* align_move: XY 到 Target 停原地 (Done 不回零) — 守卫: Z门+遮光上位+板区软限位窗 *)
				CASE alignstep OF
					0:
						刮板轴10ZDATE.xMoveAbs:=FALSE;   (* 照 A10_init step5 惯例: 先清三轴残留 xMoveAbs *)
						刮板轴9XDATE.xMoveAbs:=FALSE;
						拍照轴8YDATE.xMoveAbs:=FALSE;
						IF NOT (刮板轴10ZDATE.fActPos < ALIGN_Z_XY_GATE) THEN
							PhotoScrape_L2_ErrorCode := 421;   (* Z 非零位禁 XY 移动; 先 align_z(0) 抬起 *)
							alignstep := 0;
							bActionError := TRUE;
						ELSIF NOT 刮板拍照遮光气缸上位 THEN
							PhotoScrape_L2_ErrorCode := 425;   (* 遮光未上位: 8Y 硬互锁不放行, 先 cam_photohome(35) *)
							alignstep := 0;
							bActionError := TRUE;
						ELSE
							(* Target 与 g_sx/g_sy 同帧; 帧变换占位=恒等, 上机核实后回填 K/O (worklog C2) *)
							align_tx := ALIGN_FRAME_KX * PhotoScrape_Align_TargetX + ALIGN_FRAME_OX;
							align_ty := ALIGN_FRAME_KY * PhotoScrape_Align_TargetY + ALIGN_FRAME_OY;
							IF align_tx < ALIGN_X_WIN_MIN OR align_tx > ALIGN_X_WIN_MAX OR
							   align_ty < ALIGN_Y_WIN_MIN OR align_ty > ALIGN_Y_WIN_MAX THEN
								PhotoScrape_L2_ErrorCode := 422;   (* XY 目标在板区软限位窗外 (窗未实测回填前恒拒动, 安全默认) *)
								alignstep := 0;
								bActionError := TRUE;
							ELSE
								align_sav_vel_9X := 刮板轴9XDATE.fVelocity;   (* 持久速度暂存, Done 恢复 *)
								align_sav_vel_8Y := 拍照轴8YDATE.fVelocity;
								刮板轴9XDATE.fVelocity := ALIGN_VEL_XY;       (* 显式保守速度, 不靠持久值 (worklog C4) *)
								拍照轴8YDATE.fVelocity := ALIGN_VEL_XY;
								刮板轴9XDATE.fAbsTarget := align_tx;
								拍照轴8YDATE.fAbsTarget := align_ty;
								刮板轴9XDATE.xMoveAbs := TRUE;
								拍照轴8YDATE.xMoveAbs := TRUE;
								alignstep := 10;
							END_IF
						END_IF
					10:
						IF 刮板轴9XDATE.bAbMoveDone AND 拍照轴8YDATE.bAbMoveDone THEN
							刮板轴9XDATE.xMoveAbs := FALSE;
							拍照轴8YDATE.xMoveAbs := FALSE;
							刮板轴9XDATE.fVelocity := align_sav_vel_9X;   (* Reset 中止时不恢复=留保守慢速, 安全方向 *)
							拍照轴8YDATE.fVelocity := align_sav_vel_8Y;
							alignstep := 0;
							bActionDone := TRUE;   (* 停在原地, 不回零 *)
						END_IF
				END_CASE

			43: (* align_home: Z 先归 0 (开 XY 门) -> 9X→335 (工位停放位, 非机床零; worklog Q3) -> 8Y→0; 照 A10_init MoveAbsolute 惯例, 不走 MC_Home *)
				CASE alignstep OF
					0:
						刮板轴10ZDATE.xMoveAbs:=FALSE;
						刮板轴9XDATE.xMoveAbs:=FALSE;
						拍照轴8YDATE.xMoveAbs:=FALSE;
						IF NOT 刮板拍照遮光气缸上位 THEN
							PhotoScrape_L2_ErrorCode := 425;   (* 遮光未上位: 8Y 回零会被硬互锁挂死; 先 cam_photohome(35) *)
							alignstep := 0;
							bActionError := TRUE;
						ELSE
							alignstep := 5;
						END_IF
					5:  (* Z 已在 0 时 MoveAbsolute(0) 快速完成, 语义同"不在0先升" *)
						刮板轴10ZDATE.fAbsTarget := 0;
						刮板轴10ZDATE.xMoveAbs := TRUE;
						IF 刮板轴10ZDATE.bAbMoveDone THEN
							刮板轴10ZDATE.xMoveAbs := FALSE;
							alignstep := 10;
						END_IF
					10:
						刮板轴9XDATE.fAbsTarget := 335;
						刮板轴9XDATE.xMoveAbs := TRUE;
						IF 刮板轴9XDATE.bAbMoveDone THEN
							刮板轴9XDATE.xMoveAbs := FALSE;
							alignstep := 20;
						END_IF
					20: (* 8Y 硬互锁(遮光上位 AND Z<6)此时均满足 *)
						IF 刮板拍照遮光气缸上位 THEN
							拍照轴8YDATE.fAbsTarget := 0;
							拍照轴8YDATE.xMoveAbs := TRUE;
							IF 拍照轴8YDATE.bAbMoveDone THEN
								拍照轴8YDATE.xMoveAbs := FALSE;
								alignstep := 0;
								bActionDone := TRUE;
							END_IF
						END_IF
				END_CASE

			44: (* align_z: Z 两档 {0, 检查高度} 慢速; 降(Target>0)须 XY 在板区窗内; 上限 < 板面20.5 永不触板 *)
				CASE alignstep OF
					0:
						刮板轴10ZDATE.xMoveAbs:=FALSE;
						刮板轴9XDATE.xMoveAbs:=FALSE;
						拍照轴8YDATE.xMoveAbs:=FALSE;
						IF PhotoScrape_Align_TargetZ < 0.0 OR PhotoScrape_Align_TargetZ > ALIGN_Z_CHECK_MAX THEN
							PhotoScrape_L2_ErrorCode := 421;   (* Z 目标越档: 允许 [0, ALIGN_Z_CHECK_MAX] *)
							alignstep := 0;
							bActionError := TRUE;
						ELSIF PhotoScrape_Align_TargetZ > 0.0 AND
							(刮板轴9XDATE.fActPos < ALIGN_X_WIN_MIN OR 刮板轴9XDATE.fActPos > ALIGN_X_WIN_MAX OR
							 拍照轴8YDATE.fActPos < ALIGN_Y_WIN_MIN OR 拍照轴8YDATE.fActPos > ALIGN_Y_WIN_MAX) THEN
							PhotoScrape_L2_ErrorCode := 424;   (* 降 Z 前置: XY 须在板区窗内 (窗未回填前恒拒动) *)
							alignstep := 0;
							bActionError := TRUE;
						ELSE
							align_sav_vel_10Z := 刮板轴10ZDATE.fVelocity;
							刮板轴10ZDATE.fVelocity := ALIGN_VEL_Z;    (* 显式慢速缓降 (worklog C4/Q6) *)
							刮板轴10ZDATE.fAbsTarget := PhotoScrape_Align_TargetZ;
							刮板轴10ZDATE.xMoveAbs := TRUE;
							alignstep := 10;
						END_IF
					10:
						IF 刮板轴10ZDATE.bAbMoveDone THEN
							刮板轴10ZDATE.xMoveAbs := FALSE;
							刮板轴10ZDATE.fVelocity := align_sav_vel_10Z;
							alignstep := 0;
							bActionDone := TRUE;
						END_IF
				END_CASE
		END_CASE
		IF bActionDone THEN
			bActionDone              := FALSE;
			PhotoScrape_L2_CompletedSeq := PhotoScrape_L2_AcceptedSeq;
			PhotoScrape_L2_State        := 20;   (* DONE *)
		ELSIF bActionError THEN              (* 设备预条件未满足 -> 报错交上位机 *)
			bActionError             := FALSE;
			PhotoScrape_L2_Retryable    := TRUE;
			PhotoScrape_L2_CompletedSeq := PhotoScrape_L2_AcceptedSeq;
			PhotoScrape_L2_State        := 40;   (* ERROR; ErrorCode 由原子置 *)
		END_IF

	20, 30, 40, 50:  (* 终态: 等 Start 落沿或 Reset 回 IDLE *)
		IF (NOT PhotoScrape_L2_Start) OR PhotoScrape_L2_Reset THEN
			PhotoScrape_L2_State := 0;
		END_IF
END_CASE

ACTION A10_init_初始化:





CASE 初始化step OF
	0:
		刮板拍照真空自动:=FALSE;
		刮板拍照真空手动:=FALSE;
		刮板拍照无刷电机手动:=FALSE;
		刮板拍照无刷电机自动:=FALSE;
		刮板拍照定位气缸手动:=FALSE;
		刮板拍照定位气缸自动:=FALSE;
		粉末收集器定位手动:=FALSE;
		粉末收集器定位自动:=FALSE;
		刮板拍照遮光气缸手动:=FALSE;
		刮板拍照遮光气缸自动:=FALSE;
		刮板拍照旋转气缸手动:=FALSE;
		刮板拍照旋转气缸自动:=FALSE;
		刮板拍照下压气缸手动:=FALSE;
		刮板拍照下压气缸自动:=FALSE;
		
		
	
		
		拍照step:=0;
// 		机器人取物料step:=0;
		刮板收集step:=0;
		
		Camera_scraper_initialization_OK:=FALSE;
		Photo_preparation_completed_OK:=FALSE;
		Scraper_collection_completed:=FALSE;
		Robot_completes_material_retrieval:=FALSE;
		初始化step:=5;
	5:
		刮板轴10ZDATE.xMoveAbs:=FALSE;
		刮板轴9XDATE.xMoveAbs:=FALSE;
		拍照轴8YDATE.xMoveAbs:=FALSE;
		初始化step:=6;
	6:
		刮板轴10ZDATE.fAbsTarget:=0;
		刮板轴10ZDATE.xMoveAbs:=TRUE;
		IF 刮板轴10ZDATE.bAbMoveDone THEN
			刮板轴10ZDATE.xMoveAbs:=FALSE;
			初始化step:=10;
		END_IF
	10:
		刮板轴9XDATE.fAbsTarget:=335;
		刮板轴9XDATE.xMoveAbs:=TRUE;
		IF 刮板轴9XDATE.bAbMoveDone THEN
			刮板轴9XDATE.xMoveAbs:=FALSE;
			初始化step:=20;
		END_IF
	20:
		IF 刮板拍照遮光气缸上位 THEN
			拍照轴8YDATE.fAbsTarget:=0;
			拍照轴8YDATE.xMoveAbs:=TRUE;
			IF 拍照轴8YDATE.bAbMoveDone THEN
				拍照轴8YDATE.xMoveAbs:=FALSE;
				Camera_scraper_initialization_OK:=TRUE; bActionDone:=TRUE;
				初始化step:=0;
			END_IF	
		END_IF		
	
END_CASE
END_ACTION

ACTION A32_cam_定位:
(* 拍照定位气缸夹紧 (上位机已驱动机器人放板) *)
刮板拍照定位气缸自动:=PhotoScrape_CamLocate_Target;
bActionDone:=TRUE;
END_ACTION

ACTION A35_cam_回零:
(* 遮光上 + 拍照Y轴回零 (上位机已拍照完成) *)
CASE 拍照step OF
	0:
		刮板拍照遮光气缸自动:=FALSE;
		拍照step:=10;
	10:
		IF 刮板拍照遮光气缸上位 THEN
			拍照轴8YDATE.fAbsTarget:=0;
			拍照轴8YDATE.xMoveAbs:=TRUE;
			拍照step:=20;
		END_IF
	20:
		IF 拍照轴8YDATE.bAbMoveDone THEN
			拍照轴8YDATE.xMoveAbs:=FALSE;
			拍照step:=0;
			bActionDone:=TRUE;
		END_IF
END_CASE
END_ACTION

ACTION A34_cam_相机位:
(* 移到相机位 + 遮光下 (随后由上位机视觉控制器拍照) *)
CASE 拍照step OF
	0:
		IF 刮板拍照遮光气缸上位 THEN
// 			拍照轴8YDATE.fAbsTarget:=420;
			拍照轴8YDATE.fAbsTarget:=Photo_8Y_Target;
			拍照轴8YDATE.xMoveAbs:=TRUE;
			拍照step:=10;
		END_IF
	10:
		IF 拍照轴8YDATE.bAbMoveDone THEN
			拍照轴8YDATE.xMoveAbs:=FALSE;
			刮板拍照遮光气缸自动:=TRUE;
			拍照step:=20;
		END_IF
	20:
		IF 刮板拍照遮光气缸下位 THEN
			拍照step:=0;
			bActionDone:=TRUE;
		END_IF
END_CASE
END_ACTION

ACTION A33_cam_下压:
(* PhotoScrape press cylinder target: TRUE=press down, FALSE=release/up *)
IF PhotoScrape_CamPress_Target THEN
	刮板拍照下压气缸自动:=TRUE;
	bActionDone:=TRUE;
ELSE
	刮板拍照下压气缸自动:=FALSE;
	IF 刮板拍照下压气缸上位 THEN
		bActionDone:=TRUE;
	END_IF
END_IF
END_ACTION

ACTION A31_cam_移轴335:
(* 刮板X轴到放板/上料位 335 *)
刮板轴9XDATE.fAbsTarget:=335;
刮板轴9XDATE.xMoveAbs:=TRUE;
IF 刮板轴9XDATE.bAbMoveDone THEN
	刮板轴9XDATE.xMoveAbs:=FALSE;
	bActionDone:=TRUE;
END_IF
END_ACTION

ACTION A40_scrape_刮取:
(* 刮取单 pass: 上位机已写 g_pass_z 等 g_* 参数; 触发 PLC_CNC 跑一刀
   CNC启动/CNC完成 为 PLC 内部 SoftMotion 触发线 (保留); 多 pass 由上位机循环调用本动作 *)
CASE 刮板收集step OF
	0:
		刮板拍照真空自动:=TRUE;
		(* 吸粉动力: 真空阀 %QX7.2 只是通断, 吸力源是无刷电机 %QX7.3, 两者必须成对开。
		   本行在从 legacy A20_Scraper_collection_刮板收集 移植时遗漏 (那边是被注释),
		   导致刮取期间只开阀无吸力 -> 粉末飞溅。A41_scrape_收尾 侧一直有配对的 FALSE。 *)
		刮板拍照无刷电机自动:=TRUE;
		CNC启动:=TRUE;
		刮板收集step:=10;
	10:
		IF CNC完成 THEN
			CNC启动:=FALSE;
			刮板收集step:=0;
			bActionDone:=TRUE;
		END_IF
END_CASE
END_ACTION

ACTION A52_取料停旋转:
(* 取料收尾: 停旋转气缸 (上位机已驱动机器人退出取走收集器) *)
刮板拍照旋转气缸自动:=FALSE;
bActionDone:=TRUE;
END_ACTION

ACTION A51_取料松压:
(* 取料: 松下压气缸 (上位机已驱动机器人到收集器夹持位) *)
刮板拍照下压气缸自动:=FALSE;
IF 刮板拍照下压气缸上位 THEN
	bActionDone:=TRUE;
END_IF
END_ACTION

ACTION A41_scrape_收尾:
(* 刮取收尾: 关真空/电机, 旋转气缸翻转倒料; 定位释放由 locate_cylinder(FALSE) 统一处理 *)
刮板拍照真空自动:=FALSE;
刮板拍照无刷电机自动:=FALSE;
刮板拍照旋转气缸自动:=TRUE;
bActionDone:=TRUE;
END_ACTION

END_PROGRAM

// Device/Application/40_Man/Develop_TankDrain
PROGRAM Develop_TankDrain
VAR
	i: INT;                          // 循环索引
	BlowTimer: ARRAY[1..8] OF TON;   // Phase B 吹扫定时
	CapTimer: ARRAY[1..8] OF TON;    // Phase A 硬上限看门狗
	DryTimer: ARRAY[1..8] OF TON;    // Phase B' 原位干燥定时
	bDeployCommandsArmed: BOOL;
	bAnyDrainDeployRequest: BOOL;

END_VAR




A50_Expand_liquid_discharge_排液();

ACTION A50_Expand_liquid_discharge_排液:
// ══════════════════════════════════════════════════════════════
// 排液控制程序 v2 (per-tank 并行 FSM, 每扫描调用) — spec 2026-07-14 L2化迁移+原位干燥
// ══════════════════════════════════════════════════════════════
// 相位: 50 抽液 → 55 吹扫 → 56 原位干燥 → 98 DrainedIdle (阀全关/盖保持关/Done锁存)
// 时长 (LREAL 秒, Host_Computer 全局, 上位机派发 code 50 前写):
//   Tank_Drain_S     Phase A 判据: 组废液线持续走空满此时长
//   Tank_Drain_Cap_S Phase A 每缸硬上限: 同组并发被邻缸挟持时兜底, 锁存 Tank_Drain_CapHit[i]
//   Tank_Blow_S      Phase B 吹扫时长 (真空票保持不撤 — 主动贯通气流, v2 变更)
//   Tank_Dry_S       Phase B' 原位干燥时长 (0 = 一个扫描周期直通)
//   ⚠ 四个时长为共享标量而 FSM 每扫描活读入各缸 TON PT: 当前排液经 Develop_L2 单通道串行, 安全;
//     spec §8 trigger/wait 拆分(多缸并发排液)前须升级为每缸数组或启动时锁存, 否则后派发改写在途缸 PT
// 启动: Tank_Drain_Enable[i] AND Tank_State[i] ∈ {0, 40} (0=L2路径, 40=legacy路径)
//   ⚠ 与 50_action/Develop_L2 派发器 code 50 接受门 (10/90=REJECT 501) 为同一契约, 改一处必改另一处
// 盖(展缸i气缸j)本程序不再触碰: 开盖 = L2 code 31 (A31_放板缸回原点), 由主机 just-in-time 编排
// 传感器: 溶剂废液检测传感器 TRUE=废液管已走空; 按组共享 (缸1-4/5-8); 邻缸有液只会延迟判据不会伪造
// ══════════════════════════════════════════════════════════════

// ══ 急停联锁 ══
IF NOT 急停 THEN
    FOR i := 1 TO 8 DO
        IF (Tank_State[i] = 50) OR (Tank_State[i] = 55) OR (Tank_State[i] = 56) THEN
            Tank_State[i] := 90;
        END_IF
        DrainTimer[i](IN := FALSE, PT := T#0S);
        CapTimer[i](IN := FALSE, PT := T#0S);
        BlowTimer[i](IN := FALSE, PT := T#0S);
        DryTimer[i](IN := FALSE, PT := T#0S);
        大真空泵站位[i] := FALSE;
        CASE i OF
            1: 展缸1排液电池阀1自动 := FALSE; 展缸1吹气电池阀1自动 := FALSE;
            2: 展缸1排液电池阀2自动 := FALSE; 展缸1吹气电池阀2自动 := FALSE;
            3: 展缸1排液电池阀3自动 := FALSE; 展缸1吹气电池阀3自动 := FALSE;
            4: 展缸1排液电池阀4自动 := FALSE; 展缸1吹气电池阀4自动 := FALSE;
            5: 展缸2排液电池阀1自动 := FALSE; 展缸2吹气电池阀1自动 := FALSE;
            6: 展缸2排液电池阀2自动 := FALSE; 展缸2吹气电池阀2自动 := FALSE;
            7: 展缸2排液电池阀3自动 := FALSE; 展缸2吹气电池阀3自动 := FALSE;
            8: 展缸2排液电池阀4自动 := FALSE; 展缸2吹气电池阀4自动 := FALSE;
        END_CASE
    END_FOR
    大真空泵站位[0] := FALSE;
    RETURN;
END_IF










// PLC deploy tank-drain gate BEGIN
bAnyDrainDeployRequest := Tank_Drain_Enable[1] OR Tank_Drain_Enable[2]
	OR Tank_Drain_Enable[3] OR Tank_Drain_Enable[4]
	OR Tank_Drain_Enable[5] OR Tank_Drain_Enable[6]
	OR Tank_Drain_Enable[7] OR Tank_Drain_Enable[8];
IF ((NOT PLC_Ready) OR ((PLC_Deploy_State<>0) AND (PLC_Deploy_State<>30))) THEN
	bDeployCommandsArmed := FALSE;
	FOR i := 1 TO 8 DO
		DrainTimer[i](IN := FALSE, PT := T#0S);
		CapTimer[i](IN := FALSE, PT := T#0S);
		BlowTimer[i](IN := FALSE, PT := T#0S);
		DryTimer[i](IN := FALSE, PT := T#0S);
	END_FOR
	RETURN;
ELSIF NOT bDeployCommandsArmed THEN
	IF bAnyDrainDeployRequest THEN
		// Do not replay a request that appeared while maintenance was active.
		FOR i := 1 TO 8 DO
			DrainTimer[i](IN := FALSE, PT := T#0S);
			CapTimer[i](IN := FALSE, PT := T#0S);
			BlowTimer[i](IN := FALSE, PT := T#0S);
			DryTimer[i](IN := FALSE, PT := T#0S);
		END_FOR
		RETURN;
	ELSE
		bDeployCommandsArmed := TRUE;
	END_IF
END_IF
// PLC deploy tank-drain gate END

// ══ 主循环: 逐缸并行 FSM ══
FOR i := 1 TO 8 DO
    // 定时器每扫描调用 (TON 语义: IN 断开即复位, 天然实现"持续满足"判据)
    DrainTimer[i](IN := (Tank_State[i] = 50) AND (((i > 4) AND 展缸2溶剂废液检测传感器) OR ((i < 5) AND 展缸1溶剂废液检测传感器)),
                  PT := LREAL_TO_TIME(Tank_Drain_S * 1000.0));
    CapTimer[i](IN := (Tank_State[i] = 50), PT := LREAL_TO_TIME(Tank_Drain_Cap_S * 1000.0));
    BlowTimer[i](IN := (Tank_State[i] = 55), PT := LREAL_TO_TIME(Tank_Blow_S * 1000.0));
    DryTimer[i](IN := (Tank_State[i] = 56), PT := LREAL_TO_TIME(Tank_Dry_S * 1000.0));

    IF NOT Tank_Drain_Enable[i] THEN
        // ── 场景 1: PC 撤销 Enable → 复位 Done (握手) + 中止安全归位 (98 为静止终态不动) ──
        Tank_Drain_Done[i] := FALSE;
        IF (Tank_State[i] = 50) OR (Tank_State[i] = 55) OR (Tank_State[i] = 56) OR (Tank_State[i] = 90) THEN
            大真空泵站位[i] := FALSE;
            CASE i OF
                1: 展缸1排液电池阀1自动 := FALSE; 展缸1吹气电池阀1自动 := FALSE;
                2: 展缸1排液电池阀2自动 := FALSE; 展缸1吹气电池阀2自动 := FALSE;
                3: 展缸1排液电池阀3自动 := FALSE; 展缸1吹气电池阀3自动 := FALSE;
                4: 展缸1排液电池阀4自动 := FALSE; 展缸1吹气电池阀4自动 := FALSE;
                5: 展缸2排液电池阀1自动 := FALSE; 展缸2吹气电池阀1自动 := FALSE;
                6: 展缸2排液电池阀2自动 := FALSE; 展缸2吹气电池阀2自动 := FALSE;
                7: 展缸2排液电池阀3自动 := FALSE; 展缸2吹气电池阀3自动 := FALSE;
                8: 展缸2排液电池阀4自动 := FALSE; 展缸2吹气电池阀4自动 := FALSE;
            END_CASE
            Tank_State[i] := 0;
        END_IF
    ELSIF bDeployCommandsArmed AND ((Tank_State[i] = 0) OR (Tank_State[i] = 40)) THEN
        // ── 场景 2: 启动 Phase A — 拿泵票 + 开排液阀 (⚠ 启动门与派发器同契约) ──
        大真空泵站位[i] := TRUE;
        Tank_Drain_CapHit[i] := FALSE;
        CASE i OF
            1: 展缸1排液电池阀1自动 := TRUE;
            2: 展缸1排液电池阀2自动 := TRUE;
            3: 展缸1排液电池阀3自动 := TRUE;
            4: 展缸1排液电池阀4自动 := TRUE;
            5: 展缸2排液电池阀1自动 := TRUE;
            6: 展缸2排液电池阀2自动 := TRUE;
            7: 展缸2排液电池阀3自动 := TRUE;
            8: 展缸2排液电池阀4自动 := TRUE;
        END_CASE
        Tank_State[i] := 50;
    ELSIF Tank_State[i] = 50 THEN
        // ── 场景 3: Phase A 完成 — 判据满足或硬上限兜底 → 开吹气阀 (排液阀保持, 真空票保持) ──
        IF DrainTimer[i].Q OR CapTimer[i].Q THEN
            IF CapTimer[i].Q AND (NOT DrainTimer[i].Q) THEN
                Tank_Drain_CapHit[i] := TRUE;   // 判据未满足被迫进吹扫 (同组挟持/砂芯残液偏多), 上位机复盘
            END_IF
            CASE i OF
                1: 展缸1吹气电池阀1自动 := TRUE;
                2: 展缸1吹气电池阀2自动 := TRUE;
                3: 展缸1吹气电池阀3自动 := TRUE;
                4: 展缸1吹气电池阀4自动 := TRUE;
                5: 展缸2吹气电池阀1自动 := TRUE;
                6: 展缸2吹气电池阀2自动 := TRUE;
                7: 展缸2吹气电池阀3自动 := TRUE;
                8: 展缸2吹气电池阀4自动 := TRUE;
            END_CASE
            Tank_State[i] := 55;
        END_IF
    ELSIF Tank_State[i] = 55 THEN
        // ── 场景 4: Phase B 吹扫 — 气路贯通 (吹入→废液线), 真空票保持 (v2: 不再撤票) ──
        IF BlowTimer[i].Q THEN
            Tank_State[i] := 56;   // 干燥段气路与吹扫相同; Tank_Dry_S=0 时 DryTimer PT=0 下扫描即 Q
        END_IF
    ELSIF Tank_State[i] = 56 THEN
        // ── 场景 5: Phase B' 原位干燥完成 → 收尾: 关阀撤票, 盖不动, 终态 98 ──
        IF DryTimer[i].Q THEN
            大真空泵站位[i] := FALSE;
            CASE i OF
                1: 展缸1排液电池阀1自动 := FALSE; 展缸1吹气电池阀1自动 := FALSE;
                2: 展缸1排液电池阀2自动 := FALSE; 展缸1吹气电池阀2自动 := FALSE;
                3: 展缸1排液电池阀3自动 := FALSE; 展缸1吹气电池阀3自动 := FALSE;
                4: 展缸1排液电池阀4自动 := FALSE; 展缸1吹气电池阀4自动 := FALSE;
                5: 展缸2排液电池阀1自动 := FALSE; 展缸2吹气电池阀1自动 := FALSE;
                6: 展缸2排液电池阀2自动 := FALSE; 展缸2吹气电池阀2自动 := FALSE;
                7: 展缸2排液电池阀3自动 := FALSE; 展缸2吹气电池阀3自动 := FALSE;
                8: 展缸2排液电池阀4自动 := FALSE; 展缸2吹气电池阀4自动 := FALSE;
            END_CASE
            Tank_Drain_Done[i] := TRUE;
            Tank_State[i] := 98;
        END_IF
    END_IF
END_FOR
END_ACTION

END_PROGRAM

// Device/Application/50_action/Develop_L2
PROGRAM Develop_L2
VAR
	初始化step: INT;
	清洗STEP: INT;
	润洗展缸STEP: INT;
	上液step: INT;
	放硅胶板step: INT;
	润洗计数: INT;
	上液计数: INT;
	泵初始化完成: BOOL;
	bActionDone: BOOL;
	bActionError: BOOL;
	TON_0: TON;
	TON_1: TON;
	TON_2: TON;
	DrainTank: INT;
	L2_StartTrig: R_TRIG;
	R_TRIG: ARRAY[1..10] OF R_TRIG;
	TON: ARRAY[1..10] OF TON;
END_VAR

(* Develop 工位 L2 统一动作派发器
   按 Develop_L2_ActionCode 派发到纯设备原子动作 (不含机器人/相机/CNC 握手).
   Start 上升沿接受请求 -> RUNNING 每周期调用对应原子 -> bActionDone=DONE / bActionError=ERROR. *)
L2_StartTrig(CLK := Develop_L2_Start);

(* Global deployment/startup gate: reject before any physical action is dispatched. *)
IF L2_StartTrig.Q AND (Develop_L2_State=0)
	AND ((NOT PLC_Ready) OR (PLC_Deploy_State<>0)) THEN
	Develop_L2_AcceptedSeq := Develop_L2_RequestSeq;
	Develop_L2_ActiveCode := Develop_L2_ActionCode;
	Develop_L2_ErrorCode := 190;
	Develop_L2_Retryable := TRUE;
	Develop_L2_CompletedSeq := Develop_L2_RequestSeq;
	Develop_L2_State := 30;
	RETURN;
END_IF

CASE Develop_L2_State OF
	0:  (* IDLE *)
		Develop_L2_Step := 0;
		IF L2_StartTrig.Q THEN
			Develop_L2_AcceptedSeq := Develop_L2_RequestSeq;
			Develop_L2_ActiveCode  := Develop_L2_ActionCode;
			Develop_L2_ErrorCode   := 0;
			Develop_L2_Retryable   := FALSE;
			bActionDone  := FALSE;
			bActionError := FALSE;
			初始化step := 0;
			清洗STEP := 0;
			润洗展缸STEP := 0;
			上液step := 0;
			放硅胶板step := 0;
			(* 接受态定时器复位: TON 内部计时在 FB 停止被调用后冻结 (IN 无落沿不清零).
			   A26 经 402/复位中止退出后不再被调用, TON[7](抽吸超时看门狗)/TON[10](10s判据)
			   会带旧计时进入下次动作 -> 进场即"已超时"秒判 402 / 判据被空过.
			   故每次接受新动作时对 A26 判据域定时器统一清零, 保证窗口从零起算. *)
			TON_2(IN:=FALSE);
			TON[4](IN:=FALSE);
			TON[7](IN:=FALSE);
			TON[10](IN:=FALSE);
			DrainTank := Expand_Target_Tank;
			IF (DrainTank < 1) OR (DrainTank > 8) THEN
				Develop_L2_ErrorCode    := 102;  (* target tank out of range *)
				Develop_L2_Retryable    := TRUE;
				Develop_L2_CompletedSeq := Develop_L2_AcceptedSeq;
				Develop_L2_State        := 30;   (* REJECTED *)
			ELSE
				Expand_Group  := (DrainTank - 1) / 4 + 1;
				Expand_Number := (DrainTank - 1) MOD 4 + 1;
				CASE Develop_L2_ActionCode OF
					10, 20, 21, 22, 26, 31, 32:
						Develop_L2_SafeState := 0;
						Develop_L2_State     := 10;   (* RUNNING *)
					50:
						(* 接受门与 Develop_TankDrain 启动条件 {0,40} 为同一契约, 改一处必改另一处:
						   10/90 拒绝; 98/99 幂等直通; 0/40 新起排液; 50/55/56 置 Enable 无害=重挂在途 (恢复向导 reattach) *)
						IF (Tank_State[DrainTank] = 10) OR (Tank_State[DrainTank] = 90) THEN
							Develop_L2_ErrorCode    := 501;  (* 缸态不可排液 (Prepping/Error) *)
							Develop_L2_Retryable    := TRUE;
							Develop_L2_CompletedSeq := Develop_L2_AcceptedSeq;
							Develop_L2_State        := 30;   (* REJECTED *)
						ELSIF (Tank_State[DrainTank] = 98) OR (Tank_State[DrainTank] = 99) THEN
							Develop_L2_SafeState := 10;
							Develop_L2_State     := 10;   (* RUNNING; 幂等: 缸已排空 直接完成 *)
						ELSE
							Tank_Drain_Enable[DrainTank] := TRUE;
							Develop_L2_SafeState := 0;
							Develop_L2_State     := 10;   (* RUNNING *)
						END_IF
					51:
						IF (Tank_State[DrainTank] = 98) OR (Tank_State[DrainTank] = 99) OR (Tank_State[DrainTank] = 0) THEN
							Develop_L2_SafeState := 10;
							Develop_L2_State     := 10;   (* RUNNING; release is scan-local *)
						ELSE
							Develop_L2_ErrorCode    := 511;  (* only DrainedIdle(98)/legacy Done(99)/Idle(0) tank can be released *)
							Develop_L2_Retryable    := TRUE;
							Develop_L2_CompletedSeq := Develop_L2_AcceptedSeq;
							Develop_L2_State        := 30;   (* REJECTED *)
						END_IF
				ELSE
					Develop_L2_ErrorCode    := 101;  (* unknown action code *)
					Develop_L2_Retryable    := TRUE;
					Develop_L2_CompletedSeq := Develop_L2_AcceptedSeq;
					Develop_L2_State        := 30;   (* REJECTED *)
				END_CASE
			END_IF
		END_IF

	10: (* RUNNING *)
		IF Develop_L2_Reset THEN
			IF Develop_L2_ActiveCode = 50 THEN
				Tank_Drain_Enable[DrainTank] := FALSE;
			END_IF
			Develop_L2_State := 0;
			RETURN;
		END_IF   (* RUNNING reset aborts stuck action *)
		CASE Develop_L2_ActiveCode OF
			10: A10_init_初始化();
			20: A20_pipeline_清洗管路();
			21: A21_rinse_润洗展缸();
			26: A26_rinse_suction();
			22: A22_up_liquid_上液();
			31: A31_放板缸回原点();
			32: A32_放板缸到动点();
			50:
				Develop_L2_Step := Tank_State[DrainTank];
				IF Tank_State[DrainTank] = 90 THEN
					Develop_L2_ErrorCode := 502;  (* drain FSM error *)
					bActionError := TRUE;
				ELSIF (Tank_State[DrainTank] = 98) OR (Tank_State[DrainTank] = 99) OR Tank_Drain_Done[DrainTank] THEN
					Develop_L2_SafeState := 10;
					bActionDone := TRUE;
				END_IF
			51:
				Develop_L2_Step := Tank_State[DrainTank];
				IF (Tank_State[DrainTank] = 98) OR (Tank_State[DrainTank] = 99) OR (Tank_State[DrainTank] = 0) THEN
					Tank_Drain_Enable[DrainTank] := FALSE;
					Tank_Drain_Done[DrainTank] := FALSE;
					Tank_State[DrainTank] := 0;
					Develop_L2_SafeState := 10;
					bActionDone := TRUE;
				ELSE
					Develop_L2_ErrorCode := 511;
					bActionError := TRUE;
				END_IF
		END_CASE
		IF bActionDone THEN
			bActionDone              := FALSE;
			Develop_L2_CompletedSeq := Develop_L2_AcceptedSeq;
			Develop_L2_State        := 20;   (* DONE *)
		ELSIF bActionError THEN              (* 设备预条件未满足 -> 报错交上位机 *)
			bActionError             := FALSE;
			Develop_L2_Retryable    := TRUE;
			Develop_L2_CompletedSeq := Develop_L2_AcceptedSeq;
			Develop_L2_State        := 40;   (* ERROR; ErrorCode 由原子置 *)
		END_IF

	20, 30, 40, 50:  (* terminal: wait Start falling edge or Reset *)
		IF (NOT Develop_L2_Start) OR Develop_L2_Reset THEN
			IF Develop_L2_ActiveCode = 50 THEN  (* terminal drain cleanup *)
				Tank_Drain_Enable[DrainTank] := FALSE;
			END_IF
			Develop_L2_State := 0;
		END_IF
END_CASE

ACTION A31_放板缸回原点:
(* 放板-缸回原点 (上位机随后驱动机器人放板); 删原机器人到位/允许握手 *)
CASE Expand_Group OF
	1:
		CASE Expand_Number OF
			1:
				展缸1气缸1自动:=FALSE;
				IF 展缸1气缸1原点 THEN bActionDone:=TRUE; END_IF
			2:
				展缸1气缸2自动:=FALSE;
				IF 展缸1气缸2原点 THEN bActionDone:=TRUE; END_IF
			3:
				展缸1气缸3自动:=FALSE;
				IF 展缸1气缸3原点 THEN bActionDone:=TRUE; END_IF
			4:
				展缸1气缸4自动:=FALSE;
				IF 展缸1气缸4原点 THEN bActionDone:=TRUE; END_IF
		END_CASE
	2:
		CASE Expand_Number OF
			1:
				展缸2气缸1自动:=FALSE;
				IF 展缸2气缸1原点 THEN bActionDone:=TRUE; END_IF
			2:
				展缸2气缸2自动:=FALSE;
				IF 展缸2气缸2原点 THEN bActionDone:=TRUE; END_IF
			3:
				展缸2气缸3自动:=FALSE;
				IF 展缸2气缸3原点 THEN bActionDone:=TRUE; END_IF
			4:
				展缸2气缸4自动:=FALSE;
				IF 展缸2气缸4原点 THEN bActionDone:=TRUE; END_IF
		END_CASE
END_CASE
END_ACTION

ACTION A21_rinse_润洗展缸:
TON[1](IN:=润洗展缸STEP=15,PT:=T#0.1S);
TON_1(IN:= 润洗展缸STEP=20  , PT:=T#5S , Q=> , ET=> );
TON_2(IN:=润洗展缸STEP=30, PT:=T#3S, Q=> , ET=> );
TON[4](IN:=润洗展缸STEP=40,PT:=T#30S);
TON[10](IN:=(Expand_Group=1 AND  展缸1溶剂废液检测传感器) OR (Expand_Group=2 AND  展缸2溶剂废液检测传感器),PT:=T#10S);
R_TRIG[3](CLK:=%MX2005.5 , Q=> );  //泵空闲中



CASE 润洗展缸STEP OF
	0 :
		润洗计数:=0;
		CASE Expand_Group OF
			1:
				CASE Expand_Number OF
					1:
						展缸1进液电池阀1自动:=TRUE;
						展缸1排液电池阀1自动:=TRUE;
						展缸1气缸1自动:=TRUE;
						润洗展缸STEP:=10;
					2:
						展缸1进液电池阀2自动:=TRUE;
						展缸1排液电池阀2自动:=TRUE;
						展缸1气缸2自动:=TRUE;
						润洗展缸STEP:=10;
					3:
						展缸1进液电池阀3自动:=TRUE;
						展缸1排液电池阀3自动:=TRUE;
						展缸1气缸3自动:=TRUE;
						润洗展缸STEP:=10;
					4:
						展缸1进液电池阀4自动:=TRUE;
						展缸1排液电池阀4自动:=TRUE;
						展缸1气缸4自动:=TRUE;
						润洗展缸STEP:=10;
				END_CASE
			
			2:
				CASE Expand_Number OF
					1:
						展缸2进液电池阀1自动:=TRUE;
						展缸2排液电池阀1自动:=TRUE;
						展缸2气缸1自动:=TRUE;
						润洗展缸STEP:=10;
					2:
						展缸2进液电池阀2自动:=TRUE;
						展缸2排液电池阀2自动:=TRUE;
						展缸2气缸2自动:=TRUE;
						润洗展缸STEP:=10;
					3:
						展缸2进液电池阀3自动:=TRUE;
						展缸2排液电池阀3自动:=TRUE;
						展缸2气缸3自动:=TRUE;
						润洗展缸STEP:=10;
					4:
						展缸2进液电池阀4自动:=TRUE;
						展缸2排液电池阀4自动:=TRUE;
						展缸2气缸4自动:=TRUE;
						润洗展缸STEP:=10;
				END_CASE
		END_CASE
	10:		
		IF %MW1300=0 AND 泵站位符=FALSE  THEN
			转发转存:=Expand_forward_instructions;   
			%MW1300:=LEN(STR:= 转发转存);   //发送字节数
			泵站位符:=TRUE;
			润洗展缸STEP:=15;
		END_IF
	15:
		
		IF %MW1300=0 AND TON[1].Q THEN
			CASE Expand_Group OF
				1:
					转发转存:='/1Q$R';           //查询泵状态指令
				2:
					转发转存:='/2Q$R';           //查询泵状态指令
			END_CASE
			%MW1300:=LEN(STR:= 转发转存);
		END_IF
		
		IF R_TRIG[3].Q THEN
			泵站位符:=FALSE;
			润洗计数:=润洗计数+1;
			IF 润洗计数>=Expand_rinse_count THEN
				润洗计数:=0;
				润洗展缸STEP:=20;
			ELSE
				润洗展缸STEP:=10;
			END_IF
			
		END_IF
		
	20:
		//TON_1(IN:= TRUE  , PT:=T#5S , Q=> , ET=> );
		IF TON_1.Q THEN
			转发转存:='';
			%MW1300:=128;
			Expand_Group_clean_OK:=TRUE; bActionDone:=TRUE;
			润洗展缸STEP:=0;
		END_IF
END_CASE
END_ACTION

ACTION A20_pipeline_清洗管路:
TON[2](IN:=清洗STEP=10,PT:=T#1S);
TON_0(IN:=清洗STEP=20, PT:=T#3S , Q=> , ET=> );
R_TRIG[5](CLK:=%MX2005.5 , Q=> );  //泵空闲中
CASE 清洗STEP OF
	0 :
		IF %MW1300=0 AND 泵站位符=FALSE  THEN
			转发转存:=Expand_forward_instructions; 
			%MW1300:=LEN(STR:= 转发转存);   //发送字节数
			泵站位符:=TRUE;
			清洗STEP:=10;
		END_IF
	10:
		//TON[2](IN:=TRUE,PT:=T#1S);
		IF %MW1300=0 AND TON[2].Q THEN
			CASE Expand_Group OF
				1:
					转发转存:='/1Q$R';          //查询泵状态指令
				2:
					转发转存:='/2Q$R';          //查询泵状态指令
			END_CASE
			%MW1300:=LEN(STR:= 转发转存);
		END_IF
		
		
		IF R_TRIG[5].Q THEN
			泵站位符:=FALSE;
			清洗STEP:=20;
		END_IF
	20:
		
		IF TON_0.Q THEN
			转发转存:='';
			%MW1300:=128;
			Expand_Group_clean_OK:=TRUE; bActionDone:=TRUE;
			清洗STEP:=0;
		END_IF

		
END_CASE
END_ACTION

ACTION A32_放板缸到动点:
(* 放板-缸到动点 (上位机已驱动机器人放完板) *)
CASE Expand_Group OF
	1:
		CASE Expand_Number OF
			1:
				展缸1气缸1自动:=TRUE;
				IF 展缸1气缸1动点 THEN bActionDone:=TRUE; END_IF
			2:
				展缸1气缸2自动:=TRUE;
				IF 展缸1气缸2动点 THEN bActionDone:=TRUE; END_IF
			3:
				展缸1气缸3自动:=TRUE;
				IF 展缸1气缸3动点 THEN bActionDone:=TRUE; END_IF
			4:
				展缸1气缸4自动:=TRUE;
				IF 展缸1气缸4动点 THEN bActionDone:=TRUE; END_IF
		END_CASE
	2:
		CASE Expand_Number OF
			1:
				展缸2气缸1自动:=TRUE;
				IF 展缸2气缸1动点 THEN bActionDone:=TRUE; END_IF
			2:
				展缸2气缸2自动:=TRUE;
				IF 展缸2气缸2动点 THEN bActionDone:=TRUE; END_IF
			3:
				展缸2气缸3自动:=TRUE;
				IF 展缸2气缸3动点 THEN bActionDone:=TRUE; END_IF
			4:
				展缸2气缸4自动:=TRUE;
				IF 展缸2气缸4动点 THEN bActionDone:=TRUE; END_IF
		END_CASE
END_CASE
END_ACTION

ACTION A22_up_liquid_上液:
R_TRIG[6](CLK:=%MX2005.5 , Q=> );  //泵空闲中
TON[9](IN:=上液step=20,PT:=T#0.5S,);
IF Expand_Group>0 AND Expand_Number>0 THEN
	CASE 上液step OF
		0:
			CASE Expand_Group OF
				1:
					CASE Expand_Number OF
						1:
							展缸1进液电池阀1自动:=TRUE;
							上液step:=10;
						2:
							展缸1进液电池阀2自动:=TRUE;
							上液step:=10;
						3:
							展缸1进液电池阀3自动:=TRUE;
							上液step:=10;
						4:
							展缸1进液电池阀4自动:=TRUE;
							上液step:=10;
					END_CASE
				2:
					CASE Expand_Number OF
						1:
							展缸2进液电池阀1自动:=TRUE;
							上液step:=10;
						2:
							展缸2进液电池阀2自动:=TRUE;
							上液step:=10;
						3:
							展缸2进液电池阀3自动:=TRUE;
							上液step:=10;
						4:
							展缸2进液电池阀4自动:=TRUE;
							上液step:=10;
					END_CASE
			END_CASE
		10:
			IF %MW1300=0 AND 泵站位符=FALSE  THEN
				转发转存:=Expand_forward_instructions; 
				%MW1300:=LEN(STR:= 转发转存);   //发送字节数
				泵站位符:=TRUE;
				上液step:=20;
			END_IF
		20:
		
			IF %MW1300=0 AND TON[9].Q  THEN
				CASE Expand_Group OF
					 1:
						 转发转存:='/1Q$R';          //查询泵状态指令
					 2:
						 转发转存:='/2Q$R';          //查询泵状态指令
				END_CASE
				%MW1300:=LEN(STR:= 转发转存);
			END_IF
			
			
			IF R_TRIG[6].Q THEN
				泵站位符:=FALSE;
				转发转存:='';
				%MW1300:=128;
				上液计数:=上液计数+1;
				IF 上液计数>=Expand_up_liquid_count THEN
					上液计数:=0;
					CASE Expand_Group OF
						1:
							CASE Expand_Number OF
								1:
									展缸1进液电池阀1自动:=FALSE;
									;
								2:
									展缸1进液电池阀2自动:=FALSE;
									
								3:
									展缸1进液电池阀3自动:=FALSE;
									
								4:
									展缸1进液电池阀4自动:=FALSE;
									
							END_CASE
						2:
							CASE Expand_Number OF
								1:
									展缸2进液电池阀1自动:=FALSE;
									
								2:
									展缸2进液电池阀2自动:=FALSE;
									
								3:
									展缸2进液电池阀3自动:=FALSE;
									
								4:
									展缸2进液电池阀4自动:=FALSE;
									
							END_CASE
						END_CASE
					Expand_up_liquid_OK:=TRUE; bActionDone:=TRUE;
					上液step:=0;
				ELSE
					上液step:=10;
				END_IF
			END_IF	
    END_CASE	
END_IF
END_ACTION

ACTION A10_init_初始化:
R_TRIG[1](CLK:=%MX2005.5 , Q=> );  //泵空闲中
R_TRIG[2](CLK:=%MX2005.5 , Q=> );  //泵空闲中

CASE 初始化step OF
	0:
		润洗展缸STEP:=0;
		清洗STEP:=0;
		上液step:=0;
		放硅胶板step:=0;
// 		展开step:=0;
		expand_initialization_OK:=FALSE;
		Expand_Group_clean_OK:=FALSE;
		Expand_up_liquid_OK:=FALSE;
		Expand_silica_gel_plate_OK:=FALSE;
		CASE Expand_Group OF
			1:
				CASE Expand_Number OF
					1:
						展缸1气缸1手动:=FALSE;
						展缸1气缸1自动:=FALSE;
						展缸1进液电池阀1手动:=FALSE;
						展缸1进液电池阀1自动:=FALSE;
						展缸1排液电池阀1手动:=FALSE;
						展缸1排液电池阀1自动:=FALSE;
						展缸1吹气电池阀1手动:=FALSE;
						展缸1吹气电池阀1自动:=FALSE;
					2:
						展缸1气缸2手动:=FALSE;
						展缸1气缸2自动:=FALSE;
						展缸1进液电池阀2手动:=FALSE;
						展缸1进液电池阀2自动:=FALSE;
						展缸1排液电池阀2手动:=FALSE;
						展缸1排液电池阀2自动:=FALSE;
						展缸1吹气电池阀2手动:=FALSE;
						展缸1吹气电池阀2自动:=FALSE;	
					3:
						展缸1气缸3手动:=FALSE;
						展缸1气缸3自动:=FALSE;
						展缸1进液电池阀3手动:=FALSE;
						展缸1进液电池阀3自动:=FALSE;	
						展缸1排液电池阀3手动:=FALSE;
						展缸1排液电池阀3自动:=FALSE;
						展缸1吹气电池阀3手动:=FALSE;
						展缸1吹气电池阀3自动:=FALSE;	
					4:
						展缸1气缸4手动:=FALSE;
						展缸1气缸4自动:=FALSE;
						展缸1进液电池阀4手动:=FALSE;
						展缸1进液电池阀4自动:=FALSE;	
						展缸1排液电池阀4手动:=FALSE;
						展缸1排液电池阀4自动:=FALSE;
						展缸1吹气电池阀4手动:=FALSE;
						展缸1吹气电池阀4自动:=FALSE;	
				END_CASE
				IF %MW1300=0 AND 泵站位符=FALSE  THEN
					转发转存:='/1Z0,2,2R$R';     //泵初始化指令 
					%MW1300:=LEN(STR:= 转发转存);   //发送字节数
					泵站位符:=TRUE;
					初始化STEP:=10;
				END_IF
			2:
				CASE Expand_Number OF
					1:
						展缸2气缸1手动:=FALSE;
						展缸2气缸1自动:=FALSE;
						展缸2进液电池阀1手动:=FALSE;
						展缸2进液电池阀1自动:=FALSE;
						展缸2排液电池阀1手动:=FALSE;
						展缸2排液电池阀1自动:=FALSE;
						展缸2吹气电池阀1手动:=FALSE;
						展缸2吹气电池阀1自动:=FALSE;
					2:
						展缸2气缸2手动:=FALSE;
						展缸2气缸2自动:=FALSE;
						展缸2进液电池阀2手动:=FALSE;
						展缸2进液电池阀2自动:=FALSE;
						展缸2排液电池阀2手动:=FALSE;
						展缸2排液电池阀2自动:=FALSE;
						展缸2吹气电池阀2手动:=FALSE;
						展缸2吹气电池阀2自动:=FALSE;	
					3:
						展缸2气缸3手动:=FALSE;
						展缸2气缸3自动:=FALSE;
						展缸2进液电池阀3手动:=FALSE;
						展缸2进液电池阀3自动:=FALSE;	
						展缸2排液电池阀3手动:=FALSE;
						展缸2排液电池阀3自动:=FALSE;
						展缸2吹气电池阀3手动:=FALSE;
						展缸2吹气电池阀3自动:=FALSE;	
					4:
						展缸2气缸4手动:=FALSE;
						展缸2气缸4自动:=FALSE;
						展缸2进液电池阀4手动:=FALSE;
						展缸2进液电池阀4自动:=FALSE;	
						展缸2排液电池阀4手动:=FALSE;
						展缸2排液电池阀4自动:=FALSE;
						展缸2吹气电池阀4手动:=FALSE;
						展缸2吹气电池阀4自动:=FALSE;
				END_CASE 
				 IF %MW1300=0 AND 泵站位符=FALSE  THEN
					转发转存:='/2Z0,2,2R$R';     //泵初始化指令 
					%MW1300:=LEN(STR:= 转发转存);   //发送字节数
					泵站位符:=TRUE;
					初始化STEP:=10;
				END_IF
		END_CASE

	
		
		
	10:
		CASE Expand_Group OF
			1:
				IF %MW1300=0 THEN
					转发转存:='/1Q$R';          //查询泵状态指令
					%MW1300:=LEN(STR:= 转发转存);
				END_IF
				
				
				IF R_TRIG[1].Q THEN
					泵初始化完成:=TRUE;
					泵站位符:=FALSE;
					初始化STEP:=0; bActionDone:=TRUE;
				END_IF
			2:
				IF %MW1300=0 THEN
					转发转存:='/2Q$R';          //查询泵状态指令
					%MW1300:=LEN(STR:= 转发转存);
				END_IF
				
				IF R_TRIG[2].Q THEN
					泵初始化完成:=TRUE;
					泵站位符:=FALSE;
					初始化STEP:=0; bActionDone:=TRUE;
				END_IF
		END_CASE
END_CASE
END_ACTION

ACTION A26_rinse_suction:
(* 润洗展缸-抽吸: 真空由上位机 Pump_L2 提供 (本动作前置 vacuum_on).
   等废液抽净 -> 关进液阀/开吹气阀 -> 吹气定时 -> 关阀完成. 阀状态承接 A21_rinse 注液.
   四个时长由上位机经 Tank_Suction_* 通道写入 (派发 code 26 前落地), 免改 PLC 免下装即可调;
   变量初值 = 原硬编码值, 是通道写不进来时的唯一兜底 (PT=0 会让 TON 立即 Q). *)
TON[10](IN:=(Expand_Group=1 AND  展缸1溶剂废液检测传感器) OR (Expand_Group=2 AND  展缸2溶剂废液检测传感器),
        PT:=LREAL_TO_TIME(Tank_Suction_Empty_S * 1000.0));
TON_2(IN:=润洗展缸STEP=0, PT:=LREAL_TO_TIME(Tank_Suction_Settle_S * 1000.0));
TON[4](IN:=润洗展缸STEP=10, PT:=LREAL_TO_TIME(Tank_Suction_Blow_S * 1000.0));
TON[7](IN:=润洗展缸STEP=0, PT:=LREAL_TO_TIME(Tank_Suction_Cap_S * 1000.0));   (* 抽吸超时看门狗; 上位机 stall_timeout 须 > 本值, 否则 402 被竞态糊成"结果不明确" *)
CASE 润洗展缸STEP OF
	0:
		IF TON_2.Q THEN
			IF TON[10].Q THEN
				CASE Expand_Group OF
					1:
						CASE Expand_Number OF
							1:
								展缸1进液电池阀1自动:=FALSE;
								展缸1吹气电池阀1自动:=TRUE;
								润洗展缸STEP:=10;
							2:
								展缸1进液电池阀2自动:=FALSE;
								展缸1吹气电池阀2自动:=TRUE;
								润洗展缸STEP:=10;
							3:
								展缸1进液电池阀3自动:=FALSE;
								展缸1吹气电池阀3自动:=TRUE;
								润洗展缸STEP:=10;
							4:
								展缸1进液电池阀4自动:=FALSE;
								展缸1吹气电池阀4自动:=TRUE;
								润洗展缸STEP:=10;
						END_CASE
					2:
						CASE Expand_Number OF
							1:
								展缸2进液电池阀1自动:=FALSE;
								展缸2吹气电池阀1自动:=TRUE;
								润洗展缸STEP:=10;
							2:
								展缸2进液电池阀2自动:=FALSE;
								展缸2吹气电池阀2自动:=TRUE;
								润洗展缸STEP:=10;
							3:
								展缸2进液电池阀3自动:=FALSE;
								展缸2吹气电池阀3自动:=TRUE;
								润洗展缸STEP:=10;
							4:
								展缸2进液电池阀4自动:=FALSE;
								展缸2吹气电池阀4自动:=TRUE;
								润洗展缸STEP:=10;
						END_CASE
				END_CASE
			ELSIF TON[7].Q THEN
				Develop_L2_ErrorCode:=402;   (* 抽吸超时: 废液未抽净 *)
				润洗展缸STEP:=0;
				bActionError:=TRUE;
			END_IF
		END_IF
	10:
		IF TON[4].Q THEN
			CASE Expand_Group OF
				1:
					CASE Expand_Number OF
					1:
						展缸1排液电池阀1自动:=FALSE;
						展缸1吹气电池阀1自动:=FALSE;
						Expand_Group_clean_OK:=TRUE; bActionDone:=TRUE;
						润洗展缸STEP:=0;
					2:
						展缸1排液电池阀2自动:=FALSE;
						展缸1吹气电池阀2自动:=FALSE;
						Expand_Group_clean_OK:=TRUE; bActionDone:=TRUE;
						润洗展缸STEP:=0;
					3:
						展缸1排液电池阀3自动:=FALSE;
						展缸1吹气电池阀3自动:=FALSE;
						Expand_Group_clean_OK:=TRUE; bActionDone:=TRUE;
						润洗展缸STEP:=0;
					4:
						展缸1排液电池阀4自动:=FALSE;
						展缸1吹气电池阀4自动:=FALSE;
						Expand_Group_clean_OK:=TRUE; bActionDone:=TRUE;
						润洗展缸STEP:=0;
					END_CASE
				2:
					CASE Expand_Number OF
					1:
						展缸2排液电池阀1自动:=FALSE;
						展缸2吹气电池阀1自动:=FALSE;
						Expand_Group_clean_OK:=TRUE; bActionDone:=TRUE;
						润洗展缸STEP:=0;
					2:
						展缸2排液电池阀2自动:=FALSE;
						展缸2吹气电池阀2自动:=FALSE;
						Expand_Group_clean_OK:=TRUE; bActionDone:=TRUE;
						润洗展缸STEP:=0;
					3:
						展缸2排液电池阀3自动:=FALSE;
						展缸2吹气电池阀3自动:=FALSE;
						Expand_Group_clean_OK:=TRUE; bActionDone:=TRUE;
						润洗展缸STEP:=0;
					4:
						展缸2排液电池阀4自动:=FALSE;
						展缸2吹气电池阀4自动:=FALSE;
						Expand_Group_clean_OK:=TRUE; bActionDone:=TRUE;
						润洗展缸STEP:=0;
					END_CASE
			END_CASE
		END_IF
END_CASE
END_ACTION

END_PROGRAM

// Device/Application/50_action/Pump_L2
PROGRAM Pump_L2
VAR
	bActionDone: BOOL;
	bActionError: BOOL;
	L2_StartTrig: R_TRIG;
END_VAR

(* Pump 真空泵 L2 统一动作派发器 (独立真空泵原子动作通道).
   按 Pump_L2_ActionCode 派发: 10=真空泵开 / 20=真空泵关; 写上位机泵槽 大真空泵站位[11].
   实际线圈由 PLC_Pump_泵管理 聚合 大真空泵站位[] 驱动.
   Start 上升沿接受 -> RUNNING 调原子 -> bActionDone=DONE. *)
L2_StartTrig(CLK := Pump_L2_Start);

(* Global deployment/startup gate: reject before any physical action is dispatched. *)
IF L2_StartTrig.Q AND (Pump_L2_State=0)
	AND ((NOT PLC_Ready) OR (PLC_Deploy_State<>0)) THEN
	Pump_L2_AcceptedSeq := Pump_L2_RequestSeq;
	Pump_L2_ActiveCode := Pump_L2_ActionCode;
	Pump_L2_ErrorCode := 190;
	Pump_L2_Retryable := TRUE;
	Pump_L2_CompletedSeq := Pump_L2_RequestSeq;
	Pump_L2_State := 30;
	RETURN;
END_IF

CASE Pump_L2_State OF
	0:  (* IDLE *)
		Pump_L2_Step := 0;
		IF L2_StartTrig.Q THEN
			Pump_L2_AcceptedSeq := Pump_L2_RequestSeq;
			Pump_L2_ActiveCode  := Pump_L2_ActionCode;
			Pump_L2_ErrorCode   := 0;
			Pump_L2_Retryable   := FALSE;
			bActionDone  := FALSE;
			bActionError := FALSE;
			CASE Pump_L2_ActionCode OF
				10, 20:
					Pump_L2_SafeState := 0;
					Pump_L2_State     := 10;   (* RUNNING *)
			ELSE
				Pump_L2_ErrorCode    := 101;  (* 未知动作码 *)
				Pump_L2_Retryable    := TRUE;
				Pump_L2_CompletedSeq := Pump_L2_AcceptedSeq;
				Pump_L2_State        := 30;   (* REJECTED *)
			END_CASE
		END_IF

	10: (* RUNNING *)
		IF Pump_L2_Reset THEN                (* RUNNING 中 RESET: 中止回 IDLE *)
			Pump_L2_State := 0;
		ELSE
			CASE Pump_L2_ActiveCode OF
				10: A10_vacuum_on();
				20: A20_vacuum_off();
			END_CASE
			IF bActionDone THEN
				bActionDone          := FALSE;
				Pump_L2_CompletedSeq := Pump_L2_AcceptedSeq;
				Pump_L2_State        := 20;   (* DONE *)
			ELSIF bActionError THEN
				bActionError         := FALSE;
				Pump_L2_Retryable    := TRUE;
				Pump_L2_CompletedSeq := Pump_L2_AcceptedSeq;
				Pump_L2_State        := 40;   (* ERROR *)
			END_IF
		END_IF

	20, 30, 40, 50:  (* 终态: 等 Start 落沿或 Reset 回 IDLE *)
		IF (NOT Pump_L2_Start) OR Pump_L2_Reset THEN
			Pump_L2_State := 0;
		END_IF
END_CASE

ACTION A10_vacuum_on:
(* 真空泵开: 置上位机泵槽 (实际线圈由 PLC_Pump_泵管理 聚合 大真空泵站位[] 驱动) *)
大真空泵站位[11] := TRUE;
bActionDone := TRUE;
END_ACTION

ACTION A20_vacuum_off:
(* 真空泵关: 清上位机泵槽 (排液 [0..8] 仍可独立保持真空) *)
大真空泵站位[11] := FALSE;
bActionDone := TRUE;
END_ACTION

END_PROGRAM

// Device/Application/50_action/StagingA_L2
PROGRAM StagingA_L2
VAR
	L2_StartTrig : R_TRIG;
END_VAR

// StagingA_L2
// 功能:
//   ActionCode=24: 暂存 A 定位气缸到 Host_Computer.StagingA_LocatorA_Target
//   ActionCode=25: 暂存 B 定位气缸到 Host_Computer.StagingA_LocatorB_Target
//
// L2 State:
//   0=IDLE, 10=RUNNING, 20=DONE, 30=REJECTED, 40=ERROR, 50=INTERRUPTED
// ErrorCode:
//   0=OK, 101=BUSY, 102=DUPLICATE_SEQ, 103=UNKNOWN_ACTION, 402=RESET_INTERRUPTED

L2_StartTrig(CLK := Host_Computer.StagingA_L2_Start);

(* Global deployment/startup gate: reject before any physical action is dispatched. *)
IF L2_StartTrig.Q AND (Host_Computer.StagingA_L2_State=0)
	AND ((NOT PLC_Ready) OR (PLC_Deploy_State<>0)) THEN
	Host_Computer.StagingA_L2_AcceptedSeq := Host_Computer.StagingA_L2_RequestSeq;
	Host_Computer.StagingA_L2_ActiveCode := Host_Computer.StagingA_L2_ActionCode;
	Host_Computer.StagingA_L2_ErrorCode := 190;
	Host_Computer.StagingA_L2_Retryable := TRUE;
	Host_Computer.StagingA_L2_CompletedSeq := Host_Computer.StagingA_L2_RequestSeq;
	Host_Computer.StagingA_L2_State := 30;
	RETURN;
END_IF

// Reset: 上位机/人工复位。运行中复位给 INTERRUPTED; 非运行态复位回 IDLE。
IF Host_Computer.StagingA_L2_Reset THEN
    IF Host_Computer.StagingA_L2_State = 10 THEN
        Host_Computer.StagingA_L2_ErrorCode := 402;
        Host_Computer.StagingA_L2_Retryable := FALSE;
        Host_Computer.StagingA_L2_CompletedSeq := Host_Computer.StagingA_L2_AcceptedSeq;
        Host_Computer.StagingA_L2_State := 50;
    ELSE
        Host_Computer.StagingA_L2_State := 0;
        Host_Computer.StagingA_L2_ActiveCode := 0;
        Host_Computer.StagingA_L2_Step := 0;
        Host_Computer.StagingA_L2_ErrorCode := 0;
        Host_Computer.StagingA_L2_SafeState := 0;
        Host_Computer.StagingA_L2_Retryable := FALSE;
    END_IF
    RETURN;
END_IF

// Start 上升沿: 接受/拒绝一个请求。
IF L2_StartTrig.Q THEN
    IF Host_Computer.StagingA_L2_State <> 0 THEN
        // BUSY
        Host_Computer.StagingA_L2_ErrorCode := 101;
        Host_Computer.StagingA_L2_Retryable := TRUE;
        Host_Computer.StagingA_L2_CompletedSeq := Host_Computer.StagingA_L2_RequestSeq;
        Host_Computer.StagingA_L2_State := 30;

    ELSIF Host_Computer.StagingA_L2_RequestSeq <= Host_Computer.StagingA_L2_AcceptedSeq
       OR Host_Computer.StagingA_L2_RequestSeq <= Host_Computer.StagingA_L2_CompletedSeq THEN
        // DUPLICATE_SEQ
        Host_Computer.StagingA_L2_ErrorCode := 102;
        Host_Computer.StagingA_L2_Retryable := FALSE;
        Host_Computer.StagingA_L2_CompletedSeq := Host_Computer.StagingA_L2_RequestSeq;
        Host_Computer.StagingA_L2_State := 30;

    ELSE
        CASE Host_Computer.StagingA_L2_ActionCode OF
            24, 25:
                Host_Computer.StagingA_L2_ActiveCode := Host_Computer.StagingA_L2_ActionCode;
                Host_Computer.StagingA_L2_AcceptedSeq := Host_Computer.StagingA_L2_RequestSeq;
                Host_Computer.StagingA_L2_ErrorCode := 0;
                Host_Computer.StagingA_L2_SafeState := 0;
                Host_Computer.StagingA_L2_Retryable := FALSE;
                Host_Computer.StagingA_L2_Step := 1;
                Host_Computer.StagingA_L2_State := 10;

            ELSE
                // UNKNOWN_ACTION
                Host_Computer.StagingA_L2_ErrorCode := 103;
                Host_Computer.StagingA_L2_Retryable := FALSE;
                Host_Computer.StagingA_L2_CompletedSeq := Host_Computer.StagingA_L2_RequestSeq;
                Host_Computer.StagingA_L2_State := 30;
        END_CASE
    END_IF
END_IF

// RUNNING: 目标态动作，写对应气缸输出后立即 DONE。
IF Host_Computer.StagingA_L2_State = 10 THEN
    CASE Host_Computer.StagingA_L2_ActiveCode OF
        24:
            Host_Computer.StagingA_L2_Step := 24;
            cyinder_date.粉末收集器定位自动 := Host_Computer.StagingA_LocatorA_Target;

            Host_Computer.StagingA_L2_ErrorCode := 0;
            Host_Computer.StagingA_L2_Retryable := FALSE;
            Host_Computer.StagingA_L2_CompletedSeq := Host_Computer.StagingA_L2_AcceptedSeq;
            Host_Computer.StagingA_L2_Step := 99;
            Host_Computer.StagingA_L2_State := 20;

        25:
            Host_Computer.StagingA_L2_Step := 25;
            cyinder_date.溶液收集瓶定位自动 := Host_Computer.StagingA_LocatorB_Target;

